LIN {X 0,Y 410.698,Z 448.167,A -85,B 0,C 180,E1 -10512.418,E2 -10512.418} C_VEL
LIN {X 0,Y 412.888,Z 461.606,A -85,B 0,C 180,E1 -10512.911,E2 -10512.911} C_VEL
LIN {X 0,Y 414.693,Z 474.348,A -85,B 0,C 180,E1 -10513.572,E2 -10513.572} C_VEL
LIN {X 0,Y 414.738,Z 479.778,A -85,B 0,C 180,E1 -10513.89,E2 -10513.89} C_VEL
LIN {X 0,Y 413.947,Z 492.112,A -85,B 0,C 180,E1 -10514.742,E2 -10514.742} C_VEL
LIN {X 0,Y 413.113,Z 503.369,A -85,B 0,C 180,E1 -10515.743,E2 -10515.743} C_VEL
LIN {X 0,Y 412.398,Z 514.079,A -85,B 0,C 180,E1 -10516.95,E2 -10516.95} C_VEL
LIN {X 0,Y 411.69,Z 522.971,A -85,B 0,C 180,E1 -10518.179,E2 -10518.179} C_VEL
LIN {X 0,Y 411.063,Z 531.654,A -85,B 0,C 180,E1 -10519.658,E2 -10519.658} C_VEL
LIN {X 0,Y 410.622,Z 538.602,A -85,B 0,C 180,E1 -10521.139,E2 -10521.139} C_VEL
LIN {X 0,Y 410.285,Z 544.173,A -85,B 0,C 180,E1 -10522.619,E2 -10522.619} C_VEL
LIN {X 0,Y 410.107,Z 548.549,A -85,B 0,C 180,E1 -10524.098,E2 -10524.098} C_VEL
LIN {X 0,Y 410.096,Z 550.87,A -85,B 0,C 180,E1 -10525.084,E2 -10525.084} C_VEL
LIN {X 0,Y 409.955,Z 552.745,A -85,B 0,C 180,E1 -10526.068,E2 -10526.068} C_VEL
LIN {X 0,Y 410.007,Z 554.16,A -85,B 0,C 180,E1 -10527.052,E2 -10527.052} C_VEL
LIN {X 0,Y 409.988,Z 555.167,A -85,B 0,C 180,E1 -10528.035,E2 -10528.035} C_VEL
LIN {X 0,Y 409.959,Z 555.78,A -85,B 0,C 180,E1 -10529.018,E2 -10529.018} C_VEL
LIN {X 0,Y 409.967,Z 555.999,A -85,B 0,C 180,E1 -10530,E2 -10530} C_VEL
LIN {X 0,Y 409.959,Z 555.781,A -85,B 0,C 180,E1 -10530.982,E2 -10530.982} C_VEL
LIN {X 0,Y 409.988,Z 555.169,A -85,B 0,C 180,E1 -10531.965,E2 -10531.965} C_VEL
LIN {X 0,Y 410.007,Z 554.163,A -85,B 0,C 180,E1 -10532.948,E2 -10532.948} C_VEL
LIN {X 0,Y 409.955,Z 552.749,A -85,B 0,C 180,E1 -10533.932,E2 -10533.932} C_VEL
LIN {X 0,Y 410.108,Z 549.79,A -85,B 0,C 180,E1 -10535.408,E2 -10535.408} C_VEL
LIN {X 0,Y 410.198,Z 545.778,A -85,B 0,C 180,E1 -10536.888,E2 -10536.888} C_VEL
LIN {X 0,Y 410.551,Z 539.622,A -85,B 0,C 180,E1 -10538.615,E2 -10538.615} C_VEL
LIN {X 0,Y 410.993,Z 532.901,A -85,B 0,C 180,E1 -10540.095,E2 -10540.095} C_VEL
LIN {X 0,Y 411.585,Z 524.569,A -85,B 0,C 180,E1 -10541.574,E2 -10541.574} C_VEL
LIN {X 0,Y 412.248,Z 516.038,A -85,B 0,C 180,E1 -10542.804,E2 -10542.804} C_VEL
LIN {X 0,Y 412.983,Z 505.186,A -85,B 0,C 180,E1 -10544.068,E2 -10544.068} C_VEL
LIN {X 0,Y 413.797,Z 493.656,A -85,B 0,C 180,E1 -10545.137,E2 -10545.137} C_VEL
LIN {X 0,Y 414.677,Z 481.764,A -85,B 0,C 180,E1 -10545.986,E2 -10545.986} C_VEL
LIN {X 0,Y 414.863,Z 475.472,A -85,B 0,C 180,E1 -10546.358,E2 -10546.358} C_VEL
LIN {X 0,Y 412.982,Z 462.163,A -85,B 0,C 180,E1 -10547.062,E2 -10547.062} C_VEL
LIN {X 0,Y 410.941,Z 449.743,A -85,B 0,C 180,E1 -10547.537,E2 -10547.537} C_VEL
LIN {X 0,Y 410.707,Z 447.89,A -85,B 0,C 180,E1 -10547.606,E2 -10547.606} C_VEL
LIN {X 0,Y 411.107,Z 439.39,A -85,B 0,C 180,E1 -10551.039,E2 -10551.039} C_VEL
LIN {X 0,Y 411.526,Z 431.551,A -85,B 0,C 180,E1 -10554.197,E2 -10554.197} C_VEL
LIN {X 0,Y 412.048,Z 423.353,A -85,B 0,C 180,E1 -10557.51,E2 -10557.51} C_VEL
LIN {X 0,Y 412.657,Z 414.499,A -85,B 0,C 180,E1 -10561.185,E2 -10561.185} C_VEL
LIN {X 0,Y 413.314,Z 406.352,A -85,B 0,C 180,E1 -10564.725,E2 -10564.725} C_VEL
LIN {X 0,Y 413.431,Z 402.437,A -85,B 0,C 180,E1 -10566.511,E2 -10566.511} C_VEL
LIN {X 0,Y 412.649,Z 397.214,A -85,B 0,C 180,E1 -10569.062,E2 -10569.062} C_VEL
LIN {X 0,Y 411.729,Z 392.058,A -85,B 0,C 180,E1 -10571.737,E2 -10571.737} C_VEL
LIN {X 0,Y 411.206,Z 389.271,A -85,B 0,C 180,E1 -10573.298,E2 -10573.298} C_VEL
LIN {X 0,Y 411.175,Z 389.269,A -85,B 0,C 180,E1 -10576.866,E2 -10576.866} C_VEL
LIN {X 0,Y 411.221,Z 389.266,A -85,B 0,C 180,E1 -10580.271,E2 -10580.271} C_VEL
LIN {X 0,Y 411.198,Z 389.264,A -85,B 0,C 180,E1 -10583.447,E2 -10583.447} C_VEL
LIN {X 0,Y 411.209,Z 389.265,A -85,B 0,C 180,E1 -10586.873,E2 -10586.873} C_VEL
LIN {X 0,Y 411.235,Z 389.261,A -85,B 0,C 180,E1 -10590.644,E2 -10590.644} C_VEL
LIN {X 0,Y 411.24,Z 389.257,A -85,B 0,C 180,E1 -10593.619,E2 -10593.619} C_VEL
LIN {X 0,Y 411.205,Z 389.265,A -85,B 0,C 180,E1 -10596.853,E2 -10596.853} C_VEL
LIN {X 0,Y 411.218,Z 389.261,A -85,B 0,C 180,E1 -10600.05,E2 -10600.05} C_VEL
LIN {X 0,Y 411.266,Z 389.254,A -85,B 0,C 180,E1 -10603.131,E2 -10603.131} C_VEL
LIN {X 0,Y 411.317,Z 389.25,A -85,B 0,C 180,E1 -10606.891,E2 -10606.891} C_VEL
LIN {X 0,Y 411.311,Z 389.252,A -85,B 0,C 180,E1 -10610.162,E2 -10610.162} C_VEL
LIN {X 0,Y 411.464,Z 389.23,A -85,B 0,C 180,E1 -10613.133,E2 -10613.133} C_VEL
LIN {X 0,Y 411.313,Z 389.248,A -85,B 0,C 180,E1 -10615.099,E2 -10615.099} C_VEL
LIN {X 0,Y 411.515,Z 389.225,A -85,B 0,C 180,E1 -10618.043,E2 -10618.043} C_VEL
LIN {X 0,Y 411.646,Z 389.209,A -85,B 0,C 180,E1 -10620,E2 -10620} C_VEL
LIN {X 0,Y 411.46,Z 389.231,A -85,B 0,C 180,E1 -10622.937,E2 -10622.937} C_VEL
LIN {X 0,Y 411.464,Z 389.23,A -85,B 0,C 180,E1 -10626.867,E2 -10626.867} C_VEL
LIN {X 0,Y 411.295,Z 389.252,A -85,B 0,C 180,E1 -10629.839,E2 -10629.839} C_VEL
LIN {X 0,Y 411.309,Z 389.248,A -85,B 0,C 180,E1 -10633.104,E2 -10633.104} C_VEL
LIN {X 0,Y 411.266,Z 389.254,A -85,B 0,C 180,E1 -10636.869,E2 -10636.869} C_VEL
LIN {X 0,Y 411.234,Z 389.262,A -85,B 0,C 180,E1 -10639.987,E2 -10639.987} C_VEL
LIN {X 0,Y 411.199,Z 389.261,A -85,B 0,C 180,E1 -10643.148,E2 -10643.148} C_VEL
LIN {X 0,Y 411.24,Z 389.259,A -85,B 0,C 180,E1 -10646.381,E2 -10646.381} C_VEL
LIN {X 0,Y 411.203,Z 389.266,A -85,B 0,C 180,E1 -10649.713,E2 -10649.713} C_VEL
LIN {X 0,Y 411.209,Z 389.261,A -85,B 0,C 180,E1 -10653.156,E2 -10653.156} C_VEL
LIN {X 0,Y 411.198,Z 389.262,A -85,B 0,C 180,E1 -10656.553,E2 -10656.553} C_VEL
LIN {X 0,Y 411.221,Z 389.264,A -85,B 0,C 180,E1 -10659.729,E2 -10659.729} C_VEL
LIN {X 0,Y 411.176,Z 389.266,A -85,B 0,C 180,E1 -10663.134,E2 -10663.134} C_VEL
LIN {X 0,Y 411.235,Z 389.262,A -85,B 0,C 180,E1 -10665.872,E2 -10665.872} C_VEL
LIN {X 0,Y 411.208,Z 389.26,A -85,B 0,C 180,E1 -10668.765,E2 -10668.765} C_VEL
LIN {X 0,Y 411.194,Z 389.265,A -85,B 0,C 180,E1 -10672.026,E2 -10672.026} C_VEL
LIN {X 0,Y 411.078,Z 389.28,A -85,B 0,C 180,E1 -10675.149,E2 -10675.149} C_VEL
LIN {X 0,Y 410.745,Z 389.323,A -85,B 0,C 180,E1 -10677.966,E2 -10677.966} C_VEL
LIN {X 0,Y 410.663,Z 389.786,A -85,B 0,C 180,E1 -10679.108,E2 -10679.108} C_VEL
LIN {X 0,Y 410.601,Z 391.828,A -85,B 0,C 180,E1 -10681.363,E2 -10681.363} C_VEL
LIN {X 0,Y 410.51,Z 394.919,A -85,B 0,C 180,E1 -10684.659,E2 -10684.659} C_VEL
LIN {X 0,Y 410.426,Z 398.086,A -85,B 0,C 180,E1 -10687.869,E2 -10687.869} C_VEL
LIN {X 0,Y 410.399,Z 401.392,A -85,B 0,C 180,E1 -10691.012,E2 -10691.012} C_VEL
LIN {X 0,Y 410.37,Z 403.05,A -85,B 0,C 180,E1 -10692.502,E2 -10692.502} C_VEL
LIN {X 0,Y 414.194,Z 417.585,A -85,B 0,C 180,E1 -10693.187,E2 -10693.187} C_VEL
LIN {X 0,Y 415.645,Z 424.633,A -85,B 0,C 180,E1 -10693.592,E2 -10693.592} C_VEL
LIN {X 0,Y 415.134,Z 436.175,A -85,B 0,C 180,E1 -10694.284,E2 -10694.284} C_VEL
LIN {X 0,Y 414.53,Z 446.816,A -85,B 0,C 180,E1 -10695.103,E2 -10695.103} C_VEL
LIN {X 0,Y 413.752,Z 458.523,A -85,B 0,C 180,E1 -10696.243,E2 -10696.243} C_VEL
LIN {X 0,Y 412.944,Z 468.466,A -85,B 0,C 180,E1 -10697.467,E2 -10697.467} C_VEL
LIN {X 0,Y 412.186,Z 478.066,A -85,B 0,C 180,E1 -10698.941,E2 -10698.941} C_VEL
LIN {X 0,Y 411.551,Z 485.722,A -85,B 0,C 180,E1 -10700.416,E2 -10700.416} C_VEL
LIN {X 0,Y 410.968,Z 492.741,A -85,B 0,C 180,E1 -10702.137,E2 -10702.137} C_VEL
LIN {X 0,Y 410.668,Z 497.411,A -85,B 0,C 180,E1 -10703.613,E2 -10703.613} C_VEL
LIN {X 0,Y 410.353,Z 500.99,A -85,B 0,C 180,E1 -10705.088,E2 -10705.088} C_VEL
LIN {X 0,Y 410.376,Z 502.829,A -85,B 0,C 180,E1 -10706.072,E2 -10706.072} C_VEL
LIN {X 0,Y 410.261,Z 504.221,A -85,B 0,C 180,E1 -10707.054,E2 -10707.054} C_VEL
LIN {X 0,Y 410.072,Z 505.825,A -85,B 0,C 180,E1 -10709.018,E2 -10709.018} C_VEL
LIN {X 0,Y 410.065,Z 506.056,A -85,B 0,C 180,E1 -10710,E2 -10710} C_VEL
LIN {X 0,Y 410.148,Z 505.287,A -85,B 0,C 180,E1 -10711.964,E2 -10711.964} C_VEL
LIN {X 0,Y 410.375,Z 502.977,A -85,B 0,C 180,E1 -10713.928,E2 -10713.928} C_VEL
LIN {X 0,Y 410.369,Z 500.144,A -85,B 0,C 180,E1 -10715.405,E2 -10715.405} C_VEL
LIN {X 0,Y 410.733,Z 495.771,A -85,B 0,C 180,E1 -10717.051,E2 -10717.051} C_VEL
LIN {X 0,Y 411.077,Z 491.298,A -85,B 0,C 180,E1 -10718.356,E2 -10718.356} C_VEL
LIN {X 0,Y 411.398,Z 487.566,A -85,B 0,C 180,E1 -10719.267,E2 -10719.267} C_VEL
LIN {X 0,Y 411.046,Z 484.473,A -85,B 0,C 180,E1 -10719.965,E2 -10719.965} C_VEL
LIN {X 0,Y 407.607,Z 476.939,A -85,B 0,C 180,E1 -10721.528,E2 -10721.528} C_VEL
LIN {X 0,Y 406.099,Z 472.057,A -85,B 0,C 180,E1 -10722.379,E2 -10722.379} C_VEL
LIN {X 0,Y 406.011,Z 469.328,A -85,B 0,C 180,E1 -10722.785,E2 -10722.785} C_VEL
LIN {X 0,Y 406.832,Z 459.768,A -85,B 0,C 180,E1 -10723.996,E2 -10723.996} C_VEL
LIN {X 0,Y 407.548,Z 449.017,A -85,B 0,C 180,E1 -10725.095,E2 -10725.095} C_VEL
LIN {X 0,Y 408.242,Z 437.93,A -85,B 0,C 180,E1 -10725.989,E2 -10725.989} C_VEL
LIN {X 0,Y 408.802,Z 426.011,A -85,B 0,C 180,E1 -10726.734,E2 -10726.734} C_VEL
LIN {X 0,Y 406.332,Z 414.61,A -85,B 0,C 180,E1 -10727.395,E2 -10727.395} C_VEL
LIN {X 0,Y 403.3,Z 403.39,A -85,B 0,C 180,E1 -10727.935,E2 -10727.935} C_VEL
LIN {X 0,Y 403.301,Z 400.758,A -85,B 0,C 180,E1 -10730.397,E2 -10730.397} C_VEL
LIN {X 0,Y 403.397,Z 397.5,A -85,B 0,C 180,E1 -10733.623,E2 -10733.623} C_VEL
LIN {X 0,Y 403.481,Z 394.342,A -85,B 0,C 180,E1 -10736.929,E2 -10736.929} C_VEL
LIN {X 0,Y 403.619,Z 391.226,A -85,B 0,C 180,E1 -10740.329,E2 -10740.329} C_VEL
LIN {X 0,Y 403.696,Z 390.202,A -85,B 0,C 180,E1 -10741.485,E2 -10741.485} C_VEL
LIN {X 0,Y 404.044,Z 390.154,A -85,B 0,C 180,E1 -10745.162,E2 -10745.162} C_VEL
LIN {X 0,Y 404.155,Z 390.144,A -85,B 0,C 180,E1 -10748.508,E2 -10748.508} C_VEL
LIN {X 0,Y 404.126,Z 390.142,A -85,B 0,C 180,E1 -10751.6,E2 -10751.6} C_VEL
LIN {X 0,Y 404.148,Z 390.144,A -85,B 0,C 180,E1 -10754.522,E2 -10754.522} C_VEL
LIN {X 0,Y 404.14,Z 390.141,A -85,B 0,C 180,E1 -10757.296,E2 -10757.296} C_VEL
LIN {X 0,Y 404.172,Z 390.14,A -85,B 0,C 180,E1 -10759.956,E2 -10759.956} C_VEL
LIN {X 0,Y 404.144,Z 390.14,A -85,B 0,C 180,E1 -10763.124,E2 -10763.124} C_VEL
LIN {X 0,Y 404.149,Z 390.145,A -85,B 0,C 180,E1 -10766.188,E2 -10766.188} C_VEL
LIN {X 0,Y 404.15,Z 390.142,A -85,B 0,C 180,E1 -10769.715,E2 -10769.715} C_VEL
LIN {X 0,Y 404.199,Z 390.134,A -85,B 0,C 180,E1 -10773.123,E2 -10773.123} C_VEL
LIN {X 0,Y 404.178,Z 390.136,A -85,B 0,C 180,E1 -10775.334,E2 -10775.334} C_VEL
LIN {X 0,Y 404.143,Z 390.142,A -85,B 0,C 180,E1 -10778.581,E2 -10778.581} C_VEL
LIN {X 0,Y 404.213,Z 390.137,A -85,B 0,C 180,E1 -10781.762,E2 -10781.762} C_VEL
LIN {X 0,Y 404.211,Z 390.132,A -85,B 0,C 180,E1 -10784.882,E2 -10784.882} C_VEL
LIN {X 0,Y 404.261,Z 390.132,A -85,B 0,C 180,E1 -10787.959,E2 -10787.959} C_VEL
LIN {X 0,Y 404.27,Z 390.124,A -85,B 0,C 180,E1 -10790.998,E2 -10790.998} C_VEL
LIN {X 0,Y 404.423,Z 390.11,A -85,B 0,C 180,E1 -10794.015,E2 -10794.015} C_VEL
LIN {X 0,Y 404.485,Z 390.102,A -85,B 0,C 180,E1 -10798.008,E2 -10798.008} C_VEL
LIN {X 0,Y 404.614,Z 390.085,A -85,B 0,C 180,E1 -10800,E2 -10800} C_VEL
LIN {X 0,Y 404.42,Z 390.106,A -85,B 0,C 180,E1 -10802.988,E2 -10802.988} C_VEL
LIN {X 0,Y 404.417,Z 390.108,A -85,B 0,C 180,E1 -10806.987,E2 -10806.987} C_VEL
LIN {X 0,Y 404.275,Z 390.126,A -85,B 0,C 180,E1 -10810.011,E2 -10810.011} C_VEL
LIN {X 0,Y 404.271,Z 390.128,A -85,B 0,C 180,E1 -10813.211,E2 -10813.211} C_VEL
LIN {X 0,Y 404.22,Z 390.133,A -85,B 0,C 180,E1 -10817.007,E2 -10817.007} C_VEL
LIN {X 0,Y 404.168,Z 390.138,A -85,B 0,C 180,E1 -10820.351,E2 -10820.351} C_VEL
LIN {X 0,Y 404.172,Z 390.141,A -85,B 0,C 180,E1 -10823.574,E2 -10823.574} C_VEL
LIN {X 0,Y 404.187,Z 390.137,A -85,B 0,C 180,E1 -10825.766,E2 -10825.766} C_VEL
LIN {X 0,Y 404.199,Z 390.133,A -85,B 0,C 180,E1 -10827.999,E2 -10827.999} C_VEL
LIN {X 0,Y 404.143,Z 390.144,A -85,B 0,C 180,E1 -10831.558,E2 -10831.558} C_VEL
LIN {X 0,Y 404.188,Z 390.14,A -85,B 0,C 180,E1 -10835.016,E2 -10835.016} C_VEL
LIN {X 0,Y 404.159,Z 390.142,A -85,B 0,C 180,E1 -10838.757,E2 -10838.757} C_VEL
LIN {X 0,Y 404.126,Z 390.149,A -85,B 0,C 180,E1 -10841.6,E2 -10841.6} C_VEL
LIN {X 0,Y 404.15,Z 390.144,A -85,B 0,C 180,E1 -10844.522,E2 -10844.522} C_VEL
LIN {X 0,Y 404.136,Z 390.161,A -85,B 0,C 180,E1 -10846.378,E2 -10846.378} C_VEL
LIN {X 0,Y 405.308,Z 396.25,A -85,B 0,C 180,E1 -10849.726,E2 -10849.726} C_VEL
LIN {X 0,Y 406.301,Z 402.228,A -85,B 0,C 180,E1 -10852.741,E2 -10852.741} C_VEL
LIN {X 0,Y 406.46,Z 405.637,A -85,B 0,C 180,E1 -10854.357,E2 -10854.357} C_VEL
LIN {X 0,Y 405.815,Z 413.944,A -85,B 0,C 180,E1 -10858.059,E2 -10858.059} C_VEL
LIN {X 0,Y 405.077,Z 423.703,A -85,B 0,C 180,E1 -10862.232,E2 -10862.232} C_VEL
LIN {X 0,Y 404.463,Z 432.528,A -85,B 0,C 180,E1 -10865.899,E2 -10865.899} C_VEL
LIN {X 0,Y 403.964,Z 441.605,A -85,B 0,C 180,E1 -10869.638,E2 -10869.638} C_VEL
LIN {X 0,Y 403.652,Z 447.525,A -85,B 0,C 180,E1 -10872.077,E2 -10872.077} C_VEL
LIN {X 0,Y 406.098,Z 462.801,A -85,B 0,C 180,E1 -10872.684,E2 -10872.684} C_VEL
LIN {X 0,Y 407.872,Z 475.756,A -85,B 0,C 180,E1 -10873.394,E2 -10873.394} C_VEL
LIN {X 0,Y 407.56,Z 485.037,A -85,B 0,C 180,E1 -10873.984,E2 -10873.984} C_VEL
LIN {X 0,Y 406.728,Z 496.091,A -85,B 0,C 180,E1 -10874.85,E2 -10874.85} C_VEL
LIN {X 0,Y 405.874,Z 507.394,A -85,B 0,C 180,E1 -10875.97,E2 -10875.97} C_VEL
LIN {X 0,Y 405.196,Z 517.417,A -85,B 0,C 180,E1 -10877.224,E2 -10877.224} C_VEL
LIN {X 0,Y 404.327,Z 527.131,A -85,B 0,C 180,E1 -10878.723,E2 -10878.723} C_VEL
LIN {X 0,Y 403.782,Z 534.88,A -85,B 0,C 180,E1 -10880.229,E2 -10880.229} C_VEL
LIN {X 0,Y 403.301,Z 542.027,A -85,B 0,C 180,E1 -10881.986,E2 -10881.986} C_VEL
LIN {X 0,Y 403.07,Z 547.241,A -85,B 0,C 180,E1 -10883.65,E2 -10883.65} C_VEL
LIN {X 0,Y 403.009,Z 550.437,A -85,B 0,C 180,E1 -10884.998,E2 -10884.998} C_VEL
LIN {X 0,Y 402.878,Z 552.313,A -85,B 0,C 180,E1 -10885.999,E2 -10885.999} C_VEL
LIN {X 0,Y 402.909,Z 553.727,A -85,B 0,C 180,E1 -10887,E2 -10887} C_VEL
LIN {X 0,Y 402.921,Z 554.736,A -85,B 0,C 180,E1 -10888.001,E2 -10888.001} C_VEL
LIN {X 0,Y 402.884,Z 555.349,A -85,B 0,C 180,E1 -10889,E2 -10889} C_VEL
LIN {X 0,Y 402.89,Z 555.568,A -85,B 0,C 180,E1 -10890,E2 -10890} C_VEL
LIN {X 0,Y 402.884,Z 555.35,A -85,B 0,C 180,E1 -10890.999,E2 -10890.999} C_VEL
LIN {X 0,Y 402.921,Z 554.738,A -85,B 0,C 180,E1 -10891.999,E2 -10891.999} C_VEL
LIN {X 0,Y 402.909,Z 553.731,A -85,B 0,C 180,E1 -10893,E2 -10893} C_VEL
LIN {X 0,Y 402.878,Z 552.317,A -85,B 0,C 180,E1 -10894.001,E2 -10894.001} C_VEL
LIN {X 0,Y 403.006,Z 549.355,A -85,B 0,C 180,E1 -10895.504,E2 -10895.504} C_VEL
LIN {X 0,Y 403.116,Z 545.343,A -85,B 0,C 180,E1 -10897.01,E2 -10897.01} C_VEL
LIN {X 0,Y 403.516,Z 539.188,A -85,B 0,C 180,E1 -10898.766,E2 -10898.766} C_VEL
LIN {X 0,Y 403.965,Z 532.465,A -85,B 0,C 180,E1 -10900.272,E2 -10900.272} C_VEL
LIN {X 0,Y 404.591,Z 524.133,A -85,B 0,C 180,E1 -10901.777,E2 -10901.777} C_VEL
LIN {X 0,Y 405.264,Z 515.6,A -85,B 0,C 180,E1 -10903.029,E2 -10903.029} C_VEL
LIN {X 0,Y 405.98,Z 505.781,A -85,B 0,C 180,E1 -10904.204,E2 -10904.204} C_VEL
LIN {X 0,Y 406.821,Z 494.653,A -85,B 0,C 180,E1 -10905.275,E2 -10905.275} C_VEL
LIN {X 0,Y 407.687,Z 483.364,A -85,B 0,C 180,E1 -10906.131,E2 -10906.131} C_VEL
LIN {X 0,Y 407.882,Z 475.734,A -85,B 0,C 180,E1 -10906.606,E2 -10906.606} C_VEL
LIN {X 0,Y 406.135,Z 462.792,A -85,B 0,C 180,E1 -10907.313,E2 -10907.313} C_VEL
LIN {X 0,Y 403.91,Z 449.366,A -85,B 0,C 180,E1 -10907.85,E2 -10907.85} C_VEL
LIN {X 0,Y 403.658,Z 447.51,A -85,B 0,C 180,E1 -10907.904,E2 -10907.904} C_VEL
LIN {X 0,Y 404.098,Z 439.017,A -85,B 0,C 180,E1 -10911.422,E2 -10911.422} C_VEL
LIN {X 0,Y 404.512,Z 431.208,A -85,B 0,C 180,E1 -10914.644,E2 -10914.644} C_VEL
LIN {X 0,Y 405.094,Z 423.257,A -85,B 0,C 180,E1 -10917.932,E2 -10917.932} C_VEL
LIN {X 0,Y 405.813,Z 413.858,A -85,B 0,C 180,E1 -10921.94,E2 -10921.94} C_VEL
LIN {X 0,Y 406.329,Z 407.41,A -85,B 0,C 180,E1 -10924.805,E2 -10924.805} C_VEL
LIN {X 0,Y 406.447,Z 403.512,A -85,B 0,C 180,E1 -10926.623,E2 -10926.623} C_VEL
LIN {X 0,Y 405.627,Z 398.163,A -85,B 0,C 180,E1 -10929.288,E2 -10929.288} C_VEL
LIN {X 0,Y 404.494,Z 391.852,A -85,B 0,C 180,E1 -10932.658,E2 -10932.658} C_VEL
LIN {X 0,Y 404.127,Z 390.155,A -85,B 0,C 180,E1 -10933.621,E2 -10933.621} C_VEL
LIN {X 0,Y 404.155,Z 390.144,A -85,B 0,C 180,E1 -10936.916,E2 -10936.916} C_VEL
LIN {X 0,Y 404.171,Z 390.141,A -85,B 0,C 180,E1 -10939.955,E2 -10939.955} C_VEL
LIN {X 0,Y 404.142,Z 390.145,A -85,B 0,C 180,E1 -10943.124,E2 -10943.124} C_VEL
LIN {X 0,Y 404.147,Z 390.141,A -85,B 0,C 180,E1 -10946.188,E2 -10946.188} C_VEL
LIN {X 0,Y 404.148,Z 390.139,A -85,B 0,C 180,E1 -10949.715,E2 -10949.715} C_VEL
LIN {X 0,Y 404.197,Z 390.137,A -85,B 0,C 180,E1 -10953.123,E2 -10953.123} C_VEL
LIN {X 0,Y 404.179,Z 390.137,A -85,B 0,C 180,E1 -10955.334,E2 -10955.334} C_VEL
LIN {X 0,Y 404.142,Z 390.145,A -85,B 0,C 180,E1 -10958.581,E2 -10958.581} C_VEL
LIN {X 0,Y 404.214,Z 390.132,A -85,B 0,C 180,E1 -10961.762,E2 -10961.762} C_VEL
LIN {X 0,Y 404.211,Z 390.135,A -85,B 0,C 180,E1 -10964.882,E2 -10964.882} C_VEL
LIN {X 0,Y 404.273,Z 390.126,A -85,B 0,C 180,E1 -10967.959,E2 -10967.959} C_VEL
LIN {X 0,Y 404.437,Z 390.107,A -85,B 0,C 180,E1 -10972.1,E2 -10972.1} C_VEL
LIN {X 0,Y 404.427,Z 390.108,A -85,B 0,C 180,E1 -10974.015,E2 -10974.015} C_VEL
LIN {X 0,Y 404.484,Z 390.1,A -85,B 0,C 180,E1 -10978.009,E2 -10978.009} C_VEL
LIN {X 0,Y 404.615,Z 390.085,A -85,B 0,C 180,E1 -10980,E2 -10980} C_VEL
LIN {X 0,Y 404.418,Z 390.107,A -85,B 0,C 180,E1 -10982.988,E2 -10982.988} C_VEL
LIN {X 0,Y 404.415,Z 390.107,A -85,B 0,C 180,E1 -10986.987,E2 -10986.987} C_VEL
LIN {X 0,Y 404.261,Z 390.13,A -85,B 0,C 180,E1 -10990.012,E2 -10990.012} C_VEL
LIN {X 0,Y 404.269,Z 390.125,A -85,B 0,C 180,E1 -10993.211,E2 -10993.211} C_VEL
LIN {X 0,Y 404.219,Z 390.132,A -85,B 0,C 180,E1 -10997.007,E2 -10997.007} C_VEL
LIN {X 0,Y 404.167,Z 390.141,A -85,B 0,C 180,E1 -11000.352,E2 -11000.352} C_VEL
LIN {X 0,Y 404.166,Z 390.139,A -85,B 0,C 180,E1 -11003.575,E2 -11003.575} C_VEL
LIN {X 0,Y 404.186,Z 390.14,A -85,B 0,C 180,E1 -11005.766,E2 -11005.766} C_VEL
LIN {X 0,Y 404.198,Z 390.138,A -85,B 0,C 180,E1 -11008,E2 -11008} C_VEL
LIN {X 0,Y 404.142,Z 390.144,A -85,B 0,C 180,E1 -11011.558,E2 -11011.558} C_VEL
LIN {X 0,Y 404.188,Z 390.135,A -85,B 0,C 180,E1 -11015.016,E2 -11015.016} C_VEL
LIN {X 0,Y 404.162,Z 390.138,A -85,B 0,C 180,E1 -11018.756,E2 -11018.756} C_VEL
LIN {X 0,Y 404.126,Z 390.148,A -85,B 0,C 180,E1 -11021.6,E2 -11021.6} C_VEL
LIN {X 0,Y 404.156,Z 390.139,A -85,B 0,C 180,E1 -11024.523,E2 -11024.523} C_VEL
LIN {X 0,Y 404.21,Z 390.135,A -85,B 0,C 180,E1 -11027.305,E2 -11027.305} C_VEL
LIN {X 0,Y 404.171,Z 390.14,A -85,B 0,C 180,E1 -11029.955,E2 -11029.955} C_VEL
LIN {X 0,Y 404.12,Z 390.146,A -85,B 0,C 180,E1 -11033.129,E2 -11033.129} C_VEL
LIN {X 0,Y 404.046,Z 390.154,A -85,B 0,C 180,E1 -11034.97,E2 -11034.97} C_VEL
LIN {X 0,Y 403.618,Z 390.211,A -85,B 0,C 180,E1 -11038.563,E2 -11038.563} C_VEL
LIN {X 0,Y 403.598,Z 392.184,A -85,B 0,C 180,E1 -11040.819,E2 -11040.819} C_VEL
LIN {X 0,Y 403.455,Z 395.275,A -85,B 0,C 180,E1 -11044.184,E2 -11044.184} C_VEL
LIN {X 0,Y 403.383,Z 398.468,A -85,B 0,C 180,E1 -11047.462,E2 -11047.462} C_VEL
LIN {X 0,Y 403.365,Z 401.809,A -85,B 0,C 180,E1 -11050.668,E2 -11050.668} C_VEL
LIN {X 0,Y 403.318,Z 403.488,A -85,B 0,C 180,E1 -11052.193,E2 -11052.193} C_VEL
LIN {X 0,Y 406.891,Z 416.983,A -85,B 0,C 180,E1 -11052.83,E2 -11052.83} C_VEL
LIN {X 0,Y 408.773,Z 425.368,A -85,B 0,C 180,E1 -11053.325,E2 -11053.325} C_VEL
LIN {X 0,Y 408.328,Z 436.612,A -85,B 0,C 180,E1 -11054.015,E2 -11054.015} C_VEL
LIN {X 0,Y 407.649,Z 447.828,A -85,B 0,C 180,E1 -11054.898,E2 -11054.898} C_VEL
LIN {X 0,Y 406.894,Z 458.958,A -85,B 0,C 180,E1 -11056.006,E2 -11056.006} C_VEL
LIN {X 0,Y 406.031,Z 468.901,A -85,B 0,C 180,E1 -11057.25,E2 -11057.25} C_VEL
LIN {X 0,Y 405.243,Z 478.5,A -85,B 0,C 180,E1 -11058.749,E2 -11058.749} C_VEL
LIN {X 0,Y 404.567,Z 486.156,A -85,B 0,C 180,E1 -11060.249,E2 -11060.249} C_VEL
LIN {X 0,Y 403.937,Z 493.175,A -85,B 0,C 180,E1 -11061.999,E2 -11061.999} C_VEL
LIN {X 0,Y 403.636,Z 497.843,A -85,B 0,C 180,E1 -11063.502,E2 -11063.502} C_VEL
LIN {X 0,Y 403.279,Z 501.424,A -85,B 0,C 180,E1 -11065.001,E2 -11065.001} C_VEL
LIN {X 0,Y 403.321,Z 503.26,A -85,B 0,C 180,E1 -11066.003,E2 -11066.003} C_VEL
LIN {X 0,Y 403.199,Z 504.653,A -85,B 0,C 180,E1 -11067.003,E2 -11067.003} C_VEL
LIN {X 0,Y 402.993,Z 506.256,A -85,B 0,C 180,E1 -11069.001,E2 -11069.001} C_VEL
LIN {X 0,Y 402.983,Z 506.488,A -85,B 0,C 180,E1 -11070,E2 -11070} C_VEL
LIN {X 0,Y 403.075,Z 505.718,A -85,B 0,C 180,E1 -11071.999,E2 -11071.999} C_VEL
LIN {X 0,Y 403.32,Z 503.407,A -85,B 0,C 180,E1 -11073.997,E2 -11073.997} C_VEL
LIN {X 0,Y 403.32,Z 500.574,A -85,B 0,C 180,E1 -11075.5,E2 -11075.5} C_VEL
LIN {X 0,Y 403.695,Z 496.422,A -85,B 0,C 180,E1 -11077.102,E2 -11077.102} C_VEL
LIN {X 0,Y 404.058,Z 491.728,A -85,B 0,C 180,E1 -11078.502,E2 -11078.502} C_VEL
LIN {X 0,Y 404.665,Z 485.447,A -85,B 0,C 180,E1 -11080.002,E2 -11080.002} C_VEL
LIN {X 0,Y 405.311,Z 477.586,A -85,B 0,C 180,E1 -11081.502,E2 -11081.502} C_VEL
LIN {X 0,Y 406.011,Z 469.328,A -85,B 0,C 180,E1 -11082.785,E2 -11082.785} C_VEL
LIN {X 0,Y 405.692,Z 465.151,A -85,B 0,C 180,E1 -11083.376,E2 -11083.376} C_VEL
LIN {X 0,Y 403.424,Z 458.187,A -85,B 0,C 180,E1 -11084.329,E2 -11084.329} C_VEL
LIN {X 0,Y 401.199,Z 450.764,A -85,B 0,C 180,E1 -11085.209,E2 -11085.209} C_VEL
LIN {X 0,Y 400.935,Z 445.857,A -85,B 0,C 180,E1 -11085.678,E2 -11085.678} C_VEL
LIN {X 0,Y 401.658,Z 435.406,A -85,B 0,C 180,E1 -11086.476,E2 -11086.476} C_VEL
LIN {X 0,Y 402.018,Z 427.154,A -85,B 0,C 180,E1 -11086.983,E2 -11086.983} C_VEL
LIN {X 0,Y 399.399,Z 415.296,A -85,B 0,C 180,E1 -11087.695,E2 -11087.695} C_VEL
LIN {X 0,Y 396.237,Z 403.83,A -85,B 0,C 180,E1 -11088.25,E2 -11088.25} C_VEL
LIN {X 0,Y 396.235,Z 401.161,A -85,B 0,C 180,E1 -11090.778,E2 -11090.778} C_VEL
LIN {X 0,Y 396.373,Z 397.878,A -85,B 0,C 180,E1 -11094.067,E2 -11094.067} C_VEL
LIN {X 0,Y 396.454,Z 394.696,A -85,B 0,C 180,E1 -11097.446,E2 -11097.446} C_VEL
LIN {X 0,Y 396.604,Z 391.531,A -85,B 0,C 180,E1 -11100.924,E2 -11100.924} C_VEL
LIN {X 0,Y 396.686,Z 391.074,A -85,B 0,C 180,E1 -11102.107,E2 -11102.107} C_VEL
LIN {X 0,Y 397.007,Z 391.029,A -85,B 0,C 180,E1 -11105.48,E2 -11105.48} C_VEL
LIN {X 0,Y 397.132,Z 391.016,A -85,B 0,C 180,E1 -11108.861,E2 -11108.861} C_VEL
LIN {X 0,Y 397.072,Z 391.026,A -85,B 0,C 180,E1 -11112.267,E2 -11112.267} C_VEL
LIN {X 0,Y 397.09,Z 391.02,A -85,B 0,C 180,E1 -11115.069,E2 -11115.069} C_VEL
LIN {X 0,Y 397.07,Z 391.025,A -85,B 0,C 180,E1 -11118.021,E2 -11118.021} C_VEL
LIN {X 0,Y 397.138,Z 391.013,A -85,B 0,C 180,E1 -11121.138,E2 -11121.138} C_VEL
LIN {X 0,Y 397.124,Z 391.018,A -85,B 0,C 180,E1 -11124.497,E2 -11124.497} C_VEL
LIN {X 0,Y 397.083,Z 391.024,A -85,B 0,C 180,E1 -11127.929,E2 -11127.929} C_VEL
LIN {X 0,Y 397.126,Z 391.015,A -85,B 0,C 180,E1 -11131.456,E2 -11131.456} C_VEL
LIN {X 0,Y 397.156,Z 391.013,A -85,B 0,C 180,E1 -11134.488,E2 -11134.488} C_VEL
LIN {X 0,Y 397.1,Z 391.022,A -85,B 0,C 180,E1 -11138.182,E2 -11138.182} C_VEL
LIN {X 0,Y 397.165,Z 391.011,A -85,B 0,C 180,E1 -11141.427,E2 -11141.427} C_VEL
LIN {X 0,Y 397.184,Z 391.008,A -85,B 0,C 180,E1 -11144.608,E2 -11144.608} C_VEL
LIN {X 0,Y 397.224,Z 391.007,A -85,B 0,C 180,E1 -11147.742,E2 -11147.742} C_VEL
LIN {X 0,Y 397.24,Z 391,A -85,B 0,C 180,E1 -11150.838,E2 -11150.838} C_VEL
LIN {X 0,Y 397.373,Z 390.988,A -85,B 0,C 180,E1 -11153.908,E2 -11153.908} C_VEL
LIN {X 0,Y 397.454,Z 390.978,A -85,B 0,C 180,E1 -11157.973,E2 -11157.973} C_VEL
LIN {X 0,Y 397.584,Z 390.961,A -85,B 0,C 180,E1 -11160,E2 -11160} C_VEL
LIN {X 0,Y 397.379,Z 390.983,A -85,B 0,C 180,E1 -11163.041,E2 -11163.041} C_VEL
LIN {X 0,Y 397.369,Z 390.986,A -85,B 0,C 180,E1 -11167.112,E2 -11167.112} C_VEL
LIN {X 0,Y 397.233,Z 391.002,A -85,B 0,C 180,E1 -11170.191,E2 -11170.191} C_VEL
LIN {X 0,Y 397.231,Z 391.006,A -85,B 0,C 180,E1 -11173.321,E2 -11173.321} C_VEL
LIN {X 0,Y 397.186,Z 391.01,A -85,B 0,C 180,E1 -11177.155,E2 -11177.155} C_VEL
LIN {X 0,Y 397.107,Z 391.018,A -85,B 0,C 180,E1 -11180.73,E2 -11180.73} C_VEL
LIN {X 0,Y 397.136,Z 391.014,A -85,B 0,C 180,E1 -11184.018,E2 -11184.018} C_VEL
LIN {X 0,Y 397.198,Z 391.01,A -85,B 0,C 180,E1 -11187.39,E2 -11187.39} C_VEL
LIN {X 0,Y 397.083,Z 391.023,A -85,B 0,C 180,E1 -11190.882,E2 -11190.882} C_VEL
LIN {X 0,Y 397.129,Z 391.015,A -85,B 0,C 180,E1 -11194.493,E2 -11194.493} C_VEL
LIN {X 0,Y 397.107,Z 391.017,A -85,B 0,C 180,E1 -11198.275,E2 -11198.275} C_VEL
LIN {X 0,Y 397.092,Z 391.023,A -85,B 0,C 180,E1 -11200.908,E2 -11200.908} C_VEL
LIN {X 0,Y 397.104,Z 391.023,A -85,B 0,C 180,E1 -11203.648,E2 -11203.648} C_VEL
LIN {X 0,Y 397.115,Z 391.062,A -85,B 0,C 180,E1 -11206.002,E2 -11206.002} C_VEL
LIN {X 0,Y 398.243,Z 397.069,A -85,B 0,C 180,E1 -11209.363,E2 -11209.363} C_VEL
LIN {X 0,Y 399.229,Z 402.864,A -85,B 0,C 180,E1 -11212.39,E2 -11212.39} C_VEL
LIN {X 0,Y 399.446,Z 407.233,A -85,B 0,C 180,E1 -11214.506,E2 -11214.506} C_VEL
LIN {X 0,Y 398.781,Z 415.117,A -85,B 0,C 180,E1 -11218.081,E2 -11218.081} C_VEL
LIN {X 0,Y 398.08,Z 424.019,A -85,B 0,C 180,E1 -11221.975,E2 -11221.975} C_VEL
LIN {X 0,Y 397.459,Z 432.183,A -85,B 0,C 180,E1 -11225.447,E2 -11225.447} C_VEL
LIN {X 0,Y 396.938,Z 441.221,A -85,B 0,C 180,E1 -11229.261,E2 -11229.261} C_VEL
LIN {X 0,Y 396.611,Z 447.16,A -85,B 0,C 180,E1 -11231.768,E2 -11231.768} C_VEL
LIN {X 0,Y 398.838,Z 460.535,A -85,B 0,C 180,E1 -11232.282,E2 -11232.282} C_VEL
LIN {X 0,Y 400.678,Z 473.868,A -85,B 0,C 180,E1 -11233.004,E2 -11233.004} C_VEL
LIN {X 0,Y 401.039,Z 479.594,A -85,B 0,C 180,E1 -11233.368,E2 -11233.368} C_VEL
LIN {X 0,Y 400.178,Z 491.248,A -85,B 0,C 180,E1 -11234.204,E2 -11234.204} C_VEL
LIN {X 0,Y 399.27,Z 502.746,A -85,B 0,C 180,E1 -11235.265,E2 -11235.265} C_VEL
LIN {X 0,Y 398.486,Z 513.323,A -85,B 0,C 180,E1 -11236.5,E2 -11236.5} C_VEL
LIN {X 0,Y 397.752,Z 522.107,A -85,B 0,C 180,E1 -11237.758,E2 -11237.758} C_VEL
LIN {X 0,Y 396.982,Z 530.784,A -85,B 0,C 180,E1 -11239.287,E2 -11239.287} C_VEL
LIN {X 0,Y 396.498,Z 537.732,A -85,B 0,C 180,E1 -11240.82,E2 -11240.82} C_VEL
LIN {X 0,Y 396.14,Z 543.305,A -85,B 0,C 180,E1 -11242.353,E2 -11242.353} C_VEL
LIN {X 0,Y 395.95,Z 547.683,A -85,B 0,C 180,E1 -11243.886,E2 -11243.886} C_VEL
LIN {X 0,Y 395.922,Z 550.005,A -85,B 0,C 180,E1 -11244.908,E2 -11244.908} C_VEL
LIN {X 0,Y 395.803,Z 551.881,A -85,B 0,C 180,E1 -11245.927,E2 -11245.927} C_VEL
LIN {X 0,Y 395.813,Z 553.295,A -85,B 0,C 180,E1 -11246.946,E2 -11246.946} C_VEL
LIN {X 0,Y 395.854,Z 554.305,A -85,B 0,C 180,E1 -11247.965,E2 -11247.965} C_VEL
LIN {X 0,Y 395.813,Z 554.918,A -85,B 0,C 180,E1 -11248.982,E2 -11248.982} C_VEL
LIN {X 0,Y 395.815,Z 555.137,A -85,B 0,C 180,E1 -11250,E2 -11250} C_VEL
LIN {X 0,Y 395.813,Z 554.919,A -85,B 0,C 180,E1 -11251.017,E2 -11251.017} C_VEL
LIN {X 0,Y 395.854,Z 554.307,A -85,B 0,C 180,E1 -11252.035,E2 -11252.035} C_VEL
LIN {X 0,Y 395.813,Z 553.297,A -85,B 0,C 180,E1 -11253.053,E2 -11253.053} C_VEL
LIN {X 0,Y 395.802,Z 551.884,A -85,B 0,C 180,E1 -11254.073,E2 -11254.073} C_VEL
LIN {X 0,Y 395.907,Z 548.92,A -85,B 0,C 180,E1 -11255.603,E2 -11255.603} C_VEL
LIN {X 0,Y 396.061,Z 544.909,A -85,B 0,C 180,E1 -11257.135,E2 -11257.135} C_VEL
LIN {X 0,Y 396.458,Z 538.752,A -85,B 0,C 180,E1 -11258.923,E2 -11258.923} C_VEL
LIN {X 0,Y 396.914,Z 532.027,A -85,B 0,C 180,E1 -11260.457,E2 -11260.457} C_VEL
LIN {X 0,Y 397.582,Z 523.695,A -85,B 0,C 180,E1 -11261.988,E2 -11261.988} C_VEL
LIN {X 0,Y 398.304,Z 515.163,A -85,B 0,C 180,E1 -11263.261,E2 -11263.261} C_VEL
LIN {X 0,Y 399.102,Z 504.865,A -85,B 0,C 180,E1 -11264.507,E2 -11264.507} C_VEL
LIN {X 0,Y 399.954,Z 494.216,A -85,B 0,C 180,E1 -11265.544,E2 -11265.544} C_VEL
LIN {X 0,Y 400.859,Z 483.018,A -85,B 0,C 180,E1 -11266.407,E2 -11266.407} C_VEL
LIN {X 0,Y 401.112,Z 477.794,A -85,B 0,C 180,E1 -11266.745,E2 -11266.745} C_VEL
LIN {X 0,Y 399.448,Z 465.095,A -85,B 0,C 180,E1 -11267.495,E2 -11267.495} C_VEL
LIN {X 0,Y 397.417,Z 452.01,A -85,B 0,C 180,E1 -11268.066,E2 -11268.066} C_VEL
LIN {X 0,Y 396.61,Z 447.109,A -85,B 0,C 180,E1 -11268.232,E2 -11268.232} C_VEL
LIN {X 0,Y 397.073,Z 438.645,A -85,B 0,C 180,E1 -11271.82,E2 -11271.82} C_VEL
LIN {X 0,Y 397.518,Z 430.86,A -85,B 0,C 180,E1 -11275.107,E2 -11275.107} C_VEL
LIN {X 0,Y 398.128,Z 422.958,A -85,B 0,C 180,E1 -11278.465,E2 -11278.465} C_VEL
LIN {X 0,Y 398.827,Z 414.303,A -85,B 0,C 180,E1 -11282.238,E2 -11282.238} C_VEL
LIN {X 0,Y 399.444,Z 407.164,A -85,B 0,C 180,E1 -11285.494,E2 -11285.494} C_VEL
LIN {X 0,Y 399.222,Z 402.845,A -85,B 0,C 180,E1 -11287.609,E2 -11287.609} C_VEL
LIN {X 0,Y 398.169,Z 396.796,A -85,B 0,C 180,E1 -11290.774,E2 -11290.774} C_VEL
LIN {X 0,Y 397.124,Z 391.026,A -85,B 0,C 180,E1 -11294.085,E2 -11294.085} C_VEL
LIN {X 0,Y 397.104,Z 391.021,A -85,B 0,C 180,E1 -11296.521,E2 -11296.521} C_VEL
LIN {X 0,Y 397.117,Z 391.022,A -85,B 0,C 180,E1 -11300.423,E2 -11300.423} C_VEL
LIN {X 0,Y 397.112,Z 391.018,A -85,B 0,C 180,E1 -11304.266,E2 -11304.266} C_VEL
LIN {X 0,Y 397.117,Z 391.02,A -85,B 0,C 180,E1 -11306.727,E2 -11306.727} C_VEL
LIN {X 0,Y 397.127,Z 391.016,A -85,B 0,C 180,E1 -11310.296,E2 -11310.296} C_VEL
LIN {X 0,Y 397.197,Z 391.01,A -85,B 0,C 180,E1 -11312.61,E2 -11312.61} C_VEL
LIN {X 0,Y 397.135,Z 391.014,A -85,B 0,C 180,E1 -11315.982,E2 -11315.982} C_VEL
LIN {X 0,Y 397.141,Z 391.013,A -85,B 0,C 180,E1 -11319.705,E2 -11319.705} C_VEL
LIN {X 0,Y 397.185,Z 391.011,A -85,B 0,C 180,E1 -11322.845,E2 -11322.845} C_VEL
LIN {X 0,Y 397.229,Z 391.006,A -85,B 0,C 180,E1 -11326.679,E2 -11326.679} C_VEL
LIN {X 0,Y 397.232,Z 391.002,A -85,B 0,C 180,E1 -11329.809,E2 -11329.809} C_VEL
LIN {X 0,Y 397.368,Z 390.987,A -85,B 0,C 180,E1 -11332.888,E2 -11332.888} C_VEL
LIN {X 0,Y 397.257,Z 391,A -85,B 0,C 180,E1 -11334.925,E2 -11334.925} C_VEL
LIN {X 0,Y 397.453,Z 390.976,A -85,B 0,C 180,E1 -11337.973,E2 -11337.973} C_VEL
LIN {X 0,Y 397.585,Z 390.96,A -85,B 0,C 180,E1 -11340,E2 -11340} C_VEL
LIN {X 0,Y 397.378,Z 390.984,A -85,B 0,C 180,E1 -11343.041,E2 -11343.041} C_VEL
LIN {X 0,Y 397.368,Z 390.984,A -85,B 0,C 180,E1 -11347.112,E2 -11347.112} C_VEL
LIN {X 0,Y 397.22,Z 391.009,A -85,B 0,C 180,E1 -11350.191,E2 -11350.191} C_VEL
LIN {X 0,Y 397.23,Z 391.002,A -85,B 0,C 180,E1 -11353.321,E2 -11353.321} C_VEL
LIN {X 0,Y 397.185,Z 391.007,A -85,B 0,C 180,E1 -11357.155,E2 -11357.155} C_VEL
LIN {X 0,Y 397.106,Z 391.017,A -85,B 0,C 180,E1 -11360.73,E2 -11360.73} C_VEL
LIN {X 0,Y 397.131,Z 391.019,A -85,B 0,C 180,E1 -11364.019,E2 -11364.019} C_VEL
LIN {X 0,Y 397.197,Z 391.007,A -85,B 0,C 180,E1 -11367.39,E2 -11367.39} C_VEL
LIN {X 0,Y 397.081,Z 391.02,A -85,B 0,C 180,E1 -11370.882,E2 -11370.882} C_VEL
LIN {X 0,Y 397.128,Z 391.015,A -85,B 0,C 180,E1 -11374.493,E2 -11374.493} C_VEL
LIN {X 0,Y 397.11,Z 391.018,A -85,B 0,C 180,E1 -11378.274,E2 -11378.274} C_VEL
LIN {X 0,Y 397.092,Z 391.019,A -85,B 0,C 180,E1 -11380.909,E2 -11380.909} C_VEL
LIN {X 0,Y 397.105,Z 391.022,A -85,B 0,C 180,E1 -11383.648,E2 -11383.648} C_VEL
LIN {X 0,Y 397.164,Z 391.01,A -85,B 0,C 180,E1 -11386.512,E2 -11386.512} C_VEL
LIN {X 0,Y 397.118,Z 391.021,A -85,B 0,C 180,E1 -11389.552,E2 -11389.552} C_VEL
LIN {X 0,Y 397.083,Z 391.02,A -85,B 0,C 180,E1 -11392.794,E2 -11392.794} C_VEL
LIN {X 0,Y 396.918,Z 391.046,A -85,B 0,C 180,E1 -11395.486,E2 -11395.486} C_VEL
LIN {X 0,Y 396.597,Z 391.085,A -85,B 0,C 180,E1 -11398.277,E2 -11398.277} C_VEL
LIN {X 0,Y 396.537,Z 392.482,A -85,B 0,C 180,E1 -11400.247,E2 -11400.247} C_VEL
LIN {X 0,Y 396.425,Z 395.632,A -85,B 0,C 180,E1 -11403.691,E2 -11403.691} C_VEL
LIN {X 0,Y 396.322,Z 399.054,A -85,B 0,C 180,E1 -11407.239,E2 -11407.239} C_VEL
LIN {X 0,Y 396.289,Z 402.208,A -85,B 0,C 180,E1 -11410.308,E2 -11410.308} C_VEL
LIN {X 0,Y 396.266,Z 403.891,A -85,B 0,C 180,E1 -11411.862,E2 -11411.862} C_VEL
LIN {X 0,Y 399.868,Z 417.218,A -85,B 0,C 180,E1 -11412.509,E2 -11412.509} C_VEL
LIN {X 0,Y 401.881,Z 426.13,A -85,B 0,C 180,E1 -11413.048,E2 -11413.048} C_VEL
LIN {X 0,Y 401.652,Z 435.694,A -85,B 0,C 180,E1 -11413.642,E2 -11413.642} C_VEL
LIN {X 0,Y 400.92,Z 446.989,A -85,B 0,C 180,E1 -11414.521,E2 -11414.521} C_VEL
LIN {X 0,Y 400.22,Z 457.546,A -85,B 0,C 180,E1 -11415.562,E2 -11415.562} C_VEL
LIN {X 0,Y 399.296,Z 467.532,A -85,B 0,C 180,E1 -11416.773,E2 -11416.773} C_VEL
LIN {X 0,Y 398.573,Z 475.991,A -85,B 0,C 180,E1 -11418.042,E2 -11418.042} C_VEL
LIN {X 0,Y 397.836,Z 484.203,A -85,B 0,C 180,E1 -11419.568,E2 -11419.568} C_VEL
LIN {X 0,Y 397.257,Z 489.823,A -85,B 0,C 180,E1 -11420.838,E2 -11420.838} C_VEL
LIN {X 0,Y 396.807,Z 495.293,A -85,B 0,C 180,E1 -11422.367,E2 -11422.367} C_VEL
LIN {X 0,Y 396.435,Z 499.585,A -85,B 0,C 180,E1 -11423.894,E2 -11423.894} C_VEL
LIN {X 0,Y 396.211,Z 501.857,A -85,B 0,C 180,E1 -11424.912,E2 -11424.912} C_VEL
LIN {X 0,Y 396.247,Z 503.693,A -85,B 0,C 180,E1 -11425.932,E2 -11425.932} C_VEL
LIN {X 0,Y 396.14,Z 505.084,A -85,B 0,C 180,E1 -11426.949,E2 -11426.949} C_VEL
LIN {X 0,Y 395.917,Z 506.687,A -85,B 0,C 180,E1 -11428.983,E2 -11428.983} C_VEL
LIN {X 0,Y 395.904,Z 506.919,A -85,B 0,C 180,E1 -11430,E2 -11430} C_VEL
LIN {X 0,Y 396.005,Z 506.148,A -85,B 0,C 180,E1 -11432.034,E2 -11432.034} C_VEL
LIN {X 0,Y 396.133,Z 505.185,A -85,B 0,C 180,E1 -11433.051,E2 -11433.051} C_VEL
LIN {X 0,Y 396.246,Z 503.838,A -85,B 0,C 180,E1 -11434.068,E2 -11434.068} C_VEL
LIN {X 0,Y 396.276,Z 501.004,A -85,B 0,C 180,E1 -11435.598,E2 -11435.598} C_VEL
LIN {X 0,Y 396.633,Z 497.141,A -85,B 0,C 180,E1 -11437.125,E2 -11437.125} C_VEL
LIN {X 0,Y 397.059,Z 492.158,A -85,B 0,C 180,E1 -11438.653,E2 -11438.653} C_VEL
LIN {X 0,Y 397.695,Z 485.876,A -85,B 0,C 180,E1 -11440.179,E2 -11440.179} C_VEL
LIN {X 0,Y 398.36,Z 478.015,A -85,B 0,C 180,E1 -11441.706,E2 -11441.706} C_VEL
LIN {X 0,Y 399.25,Z 468.226,A -85,B 0,C 180,E1 -11443.229,E2 -11443.229} C_VEL
LIN {X 0,Y 400.125,Z 458.566,A -85,B 0,C 180,E1 -11444.425,E2 -11444.425} C_VEL
LIN {X 0,Y 400.816,Z 447.756,A -85,B 0,C 180,E1 -11445.51,E2 -11445.51} C_VEL
LIN {X 0,Y 400.935,Z 445.857,A -85,B 0,C 180,E1 -11445.678,E2 -11445.678} C_VEL
LIN {X 0,Y 400.667,Z 440.793,A -85,B 0,C 180,E1 -11446.119,E2 -11446.119} C_VEL
LIN {X 0,Y 399.389,Z 435.829,A -85,B 0,C 180,E1 -11446.557,E2 -11446.557} C_VEL
LIN {X 0,Y 394.225,Z 422.453,A -85,B 0,C 180,E1 -11447.62,E2 -11447.62} C_VEL
LIN {X 0,Y 393.19,Z 418.866,A -85,B 0,C 180,E1 -11447.843,E2 -11447.843} C_VEL
LIN {X 0,Y 389.613,Z 406.129,A -85,B 0,C 180,E1 -11448.502,E2 -11448.502} C_VEL
LIN {X 0,Y 389.176,Z 404.254,A -85,B 0,C 180,E1 -11448.593,E2 -11448.593} C_VEL
LIN {X 0,Y 389.196,Z 401.564,A -85,B 0,C 180,E1 -11451.171,E2 -11451.171} C_VEL
LIN {X 0,Y 389.318,Z 398.255,A -85,B 0,C 180,E1 -11454.532,E2 -11454.532} C_VEL
LIN {X 0,Y 389.401,Z 395.051,A -85,B 0,C 180,E1 -11457.986,E2 -11457.986} C_VEL
LIN {X 0,Y 389.529,Z 392.917,A -85,B 0,C 180,E1 -11460.344,E2 -11460.344} C_VEL
LIN {X 0,Y 389.591,Z 391.959,A -85,B 0,C 180,E1 -11461.544,E2 -11461.544} C_VEL
LIN {X 0,Y 389.926,Z 391.912,A -85,B 0,C 180,E1 -11465.224,E2 -11465.224} C_VEL
LIN {X 0,Y 390.041,Z 391.897,A -85,B 0,C 180,E1 -11467.781,E2 -11467.781} C_VEL
LIN {X 0,Y 390.059,Z 391.897,A -85,B 0,C 180,E1 -11470.821,E2 -11470.821} C_VEL
LIN {X 0,Y 390.058,Z 391.896,A -85,B 0,C 180,E1 -11473.886,E2 -11473.886} C_VEL
LIN {X 0,Y 390.06,Z 391.897,A -85,B 0,C 180,E1 -11476.79,E2 -11476.79} C_VEL
LIN {X 0,Y 390.061,Z 391.895,A -85,B 0,C 180,E1 -11479.561,E2 -11479.561} C_VEL
LIN {X 0,Y 390.05,Z 391.9,A -85,B 0,C 180,E1 -11482.449,E2 -11482.449} C_VEL
LIN {X 0,Y 390.088,Z 391.896,A -85,B 0,C 180,E1 -11486.047,E2 -11486.047} C_VEL
LIN {X 0,Y 390.051,Z 391.899,A -85,B 0,C 180,E1 -11489.869,E2 -11489.869} C_VEL
LIN {X 0,Y 390.117,Z 391.887,A -85,B 0,C 180,E1 -11493.232,E2 -11493.232} C_VEL
LIN {X 0,Y 390.072,Z 391.893,A -85,B 0,C 180,E1 -11496.764,E2 -11496.764} C_VEL
LIN {X 0,Y 390.108,Z 391.894,A -85,B 0,C 180,E1 -11499.983,E2 -11499.983} C_VEL
LIN {X 0,Y 390.142,Z 391.885,A -85,B 0,C 180,E1 -11503.248,E2 -11503.248} C_VEL
LIN {X 0,Y 390.199,Z 391.878,A -85,B 0,C 180,E1 -11506.562,E2 -11506.562} C_VEL
LIN {X 0,Y 390.172,Z 391.884,A -85,B 0,C 180,E1 -11509.623,E2 -11509.623} C_VEL
LIN {X 0,Y 390.289,Z 391.866,A -85,B 0,C 180,E1 -11512.759,E2 -11512.759} C_VEL
LIN {X 0,Y 390.229,Z 391.874,A -85,B 0,C 180,E1 -11514.833,E2 -11514.833} C_VEL
LIN {X 0,Y 390.422,Z 391.854,A -85,B 0,C 180,E1 -11517.937,E2 -11517.937} C_VEL
LIN {X 0,Y 390.553,Z 391.836,A -85,B 0,C 180,E1 -11520,E2 -11520} C_VEL
LIN {X 0,Y 390.314,Z 391.864,A -85,B 0,C 180,E1 -11523.096,E2 -11523.096} C_VEL
LIN {X 0,Y 390.335,Z 391.861,A -85,B 0,C 180,E1 -11526.202,E2 -11526.202} C_VEL
LIN {X 0,Y 390.32,Z 391.863,A -85,B 0,C 180,E1 -11528.282,E2 -11528.282} C_VEL
LIN {X 0,Y 390.183,Z 391.879,A -85,B 0,C 180,E1 -11532.483,E2 -11532.483} C_VEL
LIN {X 0,Y 390.144,Z 391.888,A -85,B 0,C 180,E1 -11535.677,E2 -11535.677} C_VEL
LIN {X 0,Y 390.109,Z 391.89,A -85,B 0,C 180,E1 -11538.922,E2 -11538.922} C_VEL
LIN {X 0,Y 390.044,Z 391.897,A -85,B 0,C 180,E1 -11542.234,E2 -11542.234} C_VEL
LIN {X 0,Y 390.123,Z 391.889,A -85,B 0,C 180,E1 -11545.743,E2 -11545.743} C_VEL
LIN {X 0,Y 390.063,Z 391.899,A -85,B 0,C 180,E1 -11549.109,E2 -11549.109} C_VEL
LIN {X 0,Y 390.046,Z 391.898,A -85,B 0,C 180,E1 -11552.721,E2 -11552.721} C_VEL
LIN {X 0,Y 390.06,Z 391.895,A -85,B 0,C 180,E1 -11555.825,E2 -11555.825} C_VEL
LIN {X 0,Y 390.074,Z 391.898,A -85,B 0,C 180,E1 -11559.218,E2 -11559.218} C_VEL
LIN {X 0,Y 390.046,Z 391.904,A -85,B 0,C 180,E1 -11562.374,E2 -11562.374} C_VEL
LIN {X 0,Y 390.103,Z 392.075,A -85,B 0,C 180,E1 -11565.684,E2 -11565.684} C_VEL
LIN {X 0,Y 391.155,Z 397.82,A -85,B 0,C 180,E1 -11568.993,E2 -11568.993} C_VEL
LIN {X 0,Y 392.179,Z 403.532,A -85,B 0,C 180,E1 -11572.045,E2 -11572.045} C_VEL
LIN {X 0,Y 392.489,Z 406.984,A -85,B 0,C 180,E1 -11573.778,E2 -11573.778} C_VEL
LIN {X 0,Y 392.088,Z 412.214,A -85,B 0,C 180,E1 -11576.243,E2 -11576.243} C_VEL
LIN {X 0,Y 391.622,Z 417.449,A -85,B 0,C 180,E1 -11578.638,E2 -11578.638} C_VEL
LIN {X 0,Y 390.976,Z 425.31,A -85,B 0,C 180,E1 -11582.136,E2 -11582.136} C_VEL
LIN {X 0,Y 390.374,Z 433.13,A -85,B 0,C 180,E1 -11585.539,E2 -11585.539} C_VEL
LIN {X 0,Y 389.907,Z 440.832,A -85,B 0,C 180,E1 -11588.869,E2 -11588.869} C_VEL
LIN {X 0,Y 389.569,Z 446.744,A -85,B 0,C 180,E1 -11591.426,E2 -11591.426} C_VEL
LIN {X 0,Y 391.86,Z 460.659,A -85,B 0,C 180,E1 -11591.979,E2 -11591.979} C_VEL
LIN {X 0,Y 393.656,Z 474.09,A -85,B 0,C 180,E1 -11592.73,E2 -11592.73} C_VEL
LIN {X 0,Y 394.175,Z 479.454,A -85,B 0,C 180,E1 -11593.089,E2 -11593.089} C_VEL
LIN {X 0,Y 393.346,Z 490.819,A -85,B 0,C 180,E1 -11593.922,E2 -11593.922} C_VEL
LIN {X 0,Y 392.408,Z 501.84,A -85,B 0,C 180,E1 -11594.948,E2 -11594.948} C_VEL
LIN {X 0,Y 391.683,Z 511.49,A -85,B 0,C 180,E1 -11596.072,E2 -11596.072} C_VEL
LIN {X 0,Y 390.801,Z 521.675,A -85,B 0,C 180,E1 -11597.537,E2 -11597.537} C_VEL
LIN {X 0,Y 389.965,Z 530.35,A -85,B 0,C 180,E1 -11599.092,E2 -11599.092} C_VEL
LIN {X 0,Y 389.453,Z 537.299,A -85,B 0,C 180,E1 -11600.653,E2 -11600.653} C_VEL
LIN {X 0,Y 389.078,Z 542.872,A -85,B 0,C 180,E1 -11602.214,E2 -11602.214} C_VEL
LIN {X 0,Y 388.834,Z 548.024,A -85,B 0,C 180,E1 -11604.094,E2 -11604.094} C_VEL
LIN {X 0,Y 388.73,Z 551.45,A -85,B 0,C 180,E1 -11605.853,E2 -11605.853} C_VEL
LIN {X 0,Y 388.788,Z 553.875,A -85,B 0,C 180,E1 -11607.928,E2 -11607.928} C_VEL
LIN {X 0,Y 388.743,Z 554.488,A -85,B 0,C 180,E1 -11608.964,E2 -11608.964} C_VEL
LIN {X 0,Y 388.742,Z 554.707,A -85,B 0,C 180,E1 -11610,E2 -11610} C_VEL
LIN {X 0,Y 388.743,Z 554.488,A -85,B 0,C 180,E1 -11611.036,E2 -11611.036} C_VEL
LIN {X 0,Y 388.788,Z 553.876,A -85,B 0,C 180,E1 -11612.072,E2 -11612.072} C_VEL
LIN {X 0,Y 388.729,Z 551.452,A -85,B 0,C 180,E1 -11614.147,E2 -11614.147} C_VEL
LIN {X 0,Y 388.831,Z 548.034,A -85,B 0,C 180,E1 -11615.901,E2 -11615.901} C_VEL
LIN {X 0,Y 389.078,Z 542.867,A -85,B 0,C 180,E1 -11617.786,E2 -11617.786} C_VEL
LIN {X 0,Y 389.453,Z 537.295,A -85,B 0,C 180,E1 -11619.347,E2 -11619.347} C_VEL
LIN {X 0,Y 389.963,Z 530.344,A -85,B 0,C 180,E1 -11620.908,E2 -11620.908} C_VEL
LIN {X 0,Y 390.796,Z 521.666,A -85,B 0,C 180,E1 -11622.463,E2 -11622.463} C_VEL
LIN {X 0,Y 391.531,Z 513.09,A -85,B 0,C 180,E1 -11623.716,E2 -11623.716} C_VEL
LIN {X 0,Y 392.293,Z 503.007,A -85,B 0,C 180,E1 -11624.924,E2 -11624.924} C_VEL
LIN {X 0,Y 393.19,Z 492.344,A -85,B 0,C 180,E1 -11625.951,E2 -11625.951} C_VEL
LIN {X 0,Y 394.092,Z 481.093,A -85,B 0,C 180,E1 -11626.802,E2 -11626.802} C_VEL
LIN {X 0,Y 393.905,Z 475.967,A -85,B 0,C 180,E1 -11627.146,E2 -11627.146} C_VEL
LIN {X 0,Y 392.153,Z 462.512,A -85,B 0,C 180,E1 -11627.924,E2 -11627.924} C_VEL
LIN {X 0,Y 389.883,Z 448.784,A -85,B 0,C 180,E1 -11628.507,E2 -11628.507} C_VEL
LIN {X 0,Y 389.578,Z 446.603,A -85,B 0,C 180,E1 -11628.607,E2 -11628.607} C_VEL
LIN {X 0,Y 390.048,Z 438.263,A -85,B 0,C 180,E1 -11632.234,E2 -11632.234} C_VEL
LIN {X 0,Y 390.618,Z 429.809,A -85,B 0,C 180,E1 -11635.894,E2 -11635.894} C_VEL
LIN {X 0,Y 391.168,Z 422.64,A -85,B 0,C 180,E1 -11639.019,E2 -11639.019} C_VEL
LIN {X 0,Y 391.853,Z 414.724,A -85,B 0,C 180,E1 -11642.552,E2 -11642.552} C_VEL
LIN {X 0,Y 392.46,Z 408.231,A -85,B 0,C 180,E1 -11645.591,E2 -11645.591} C_VEL
LIN {X 0,Y 392.264,Z 404.332,A -85,B 0,C 180,E1 -11647.529,E2 -11647.529} C_VEL
LIN {X 0,Y 391.407,Z 399.148,A -85,B 0,C 180,E1 -11650.271,E2 -11650.271} C_VEL
LIN {X 0,Y 390.468,Z 394.042,A -85,B 0,C 180,E1 -11653.154,E2 -11653.154} C_VEL
LIN {X 0,Y 390.085,Z 391.904,A -85,B 0,C 180,E1 -11654.485,E2 -11654.485} C_VEL
LIN {X 0,Y 390.034,Z 391.903,A -85,B 0,C 180,E1 -11658.187,E2 -11658.187} C_VEL
LIN {X 0,Y 390.095,Z 391.896,A -85,B 0,C 180,E1 -11660.908,E2 -11660.908} C_VEL
LIN {X 0,Y 390.088,Z 391.896,A -85,B 0,C 180,E1 -11664.793,E2 -11664.793} C_VEL
LIN {X 0,Y 390.034,Z 391.898,A -85,B 0,C 180,E1 -11667.875,E2 -11667.875} C_VEL
LIN {X 0,Y 390.061,Z 391.899,A -85,B 0,C 180,E1 -11670.891,E2 -11670.891} C_VEL
LIN {X 0,Y 390.121,Z 391.889,A -85,B 0,C 180,E1 -11674.257,E2 -11674.257} C_VEL
LIN {X 0,Y 390.042,Z 391.897,A -85,B 0,C 180,E1 -11677.766,E2 -11677.766} C_VEL
LIN {X 0,Y 390.109,Z 391.89,A -85,B 0,C 180,E1 -11681.078,E2 -11681.078} C_VEL
LIN {X 0,Y 390.143,Z 391.887,A -85,B 0,C 180,E1 -11684.323,E2 -11684.323} C_VEL
LIN {X 0,Y 390.181,Z 391.879,A -85,B 0,C 180,E1 -11687.517,E2 -11687.517} C_VEL
LIN {X 0,Y 390.318,Z 391.863,A -85,B 0,C 180,E1 -11691.718,E2 -11691.718} C_VEL
LIN {X 0,Y 390.334,Z 391.861,A -85,B 0,C 180,E1 -11693.798,E2 -11693.798} C_VEL
LIN {X 0,Y 390.421,Z 391.851,A -85,B 0,C 180,E1 -11697.937,E2 -11697.937} C_VEL
LIN {X 0,Y 390.554,Z 391.836,A -85,B 0,C 180,E1 -11700,E2 -11700} C_VEL
LIN {X 0,Y 390.313,Z 391.863,A -85,B 0,C 180,E1 -11703.097,E2 -11703.097} C_VEL
LIN {X 0,Y 390.313,Z 391.864,A -85,B 0,C 180,E1 -11706.652,E2 -11706.652} C_VEL
LIN {X 0,Y 390.208,Z 391.876,A -85,B 0,C 180,E1 -11709.329,E2 -11709.329} C_VEL
LIN {X 0,Y 390.197,Z 391.878,A -85,B 0,C 180,E1 -11713.438,E2 -11713.438} C_VEL
LIN {X 0,Y 390.152,Z 391.884,A -85,B 0,C 180,E1 -11717.308,E2 -11717.308} C_VEL
LIN {X 0,Y 390.09,Z 391.893,A -85,B 0,C 180,E1 -11720.47,E2 -11720.47} C_VEL
LIN {X 0,Y 390.076,Z 391.893,A -85,B 0,C 180,E1 -11723.352,E2 -11723.352} C_VEL
LIN {X 0,Y 390.116,Z 391.888,A -85,B 0,C 180,E1 -11726.768,E2 -11726.768} C_VEL
LIN {X 0,Y 390.042,Z 391.899,A -85,B 0,C 180,E1 -11730.3,E2 -11730.3} C_VEL
LIN {X 0,Y 390.071,Z 391.898,A -85,B 0,C 180,E1 -11734.025,E2 -11734.025} C_VEL
LIN {X 0,Y 390.048,Z 391.899,A -85,B 0,C 180,E1 -11737.551,E2 -11737.551} C_VEL
LIN {X 0,Y 390.06,Z 391.895,A -85,B 0,C 180,E1 -11740.822,E2 -11740.822} C_VEL
LIN {X 0,Y 390.061,Z 391.899,A -85,B 0,C 180,E1 -11743.887,E2 -11743.887} C_VEL
LIN {X 0,Y 390.118,Z 391.887,A -85,B 0,C 180,E1 -11746.798,E2 -11746.798} C_VEL
LIN {X 0,Y 390.072,Z 391.899,A -85,B 0,C 180,E1 -11749.562,E2 -11749.562} C_VEL
LIN {X 0,Y 390.038,Z 391.897,A -85,B 0,C 180,E1 -11752.451,E2 -11752.451} C_VEL
LIN {X 0,Y 389.926,Z 391.912,A -85,B 0,C 180,E1 -11754.776,E2 -11754.776} C_VEL
LIN {X 0,Y 389.579,Z 391.959,A -85,B 0,C 180,E1 -11757.982,E2 -11757.982} C_VEL
LIN {X 0,Y 389.53,Z 391.965,A -85,B 0,C 180,E1 -11758.451,E2 -11758.451} C_VEL
LIN {X 0,Y 389.475,Z 393.888,A -85,B 0,C 180,E1 -11760.843,E2 -11760.843} C_VEL
LIN {X 0,Y 389.38,Z 397.213,A -85,B 0,C 180,E1 -11764.484,E2 -11764.484} C_VEL
LIN {X 0,Y 389.249,Z 400.35,A -85,B 0,C 180,E1 -11767.718,E2 -11767.718} C_VEL
LIN {X 0,Y 389.196,Z 403.806,A -85,B 0,C 180,E1 -11771.032,E2 -11771.032} C_VEL
LIN {X 0,Y 389.219,Z 404.31,A -85,B 0,C 180,E1 -11771.51,E2 -11771.51} C_VEL
LIN {X 0,Y 393.154,Z 418.793,A -85,B 0,C 180,E1 -11772.251,E2 -11772.251} C_VEL
LIN {X 0,Y 395.231,Z 428.918,A -85,B 0,C 180,E1 -11772.894,E2 -11772.894} C_VEL
LIN {X 0,Y 394.534,Z 440.986,A -85,B 0,C 180,E1 -11773.707,E2 -11773.707} C_VEL
LIN {X 0,Y 393.772,Z 451.57,A -85,B 0,C 180,E1 -11774.63,E2 -11774.63} C_VEL
LIN {X 0,Y 392.936,Z 461.964,A -85,B 0,C 180,E1 -11775.763,E2 -11775.763} C_VEL
LIN {X 0,Y 392.085,Z 471.535,A -85,B 0,C 180,E1 -11777.052,E2 -11777.052} C_VEL
LIN {X 0,Y 391.352,Z 479.369,A -85,B 0,C 180,E1 -11778.344,E2 -11778.344} C_VEL
LIN {X 0,Y 390.616,Z 487.023,A -85,B 0,C 180,E1 -11779.897,E2 -11779.897} C_VEL
LIN {X 0,Y 389.91,Z 494.042,A -85,B 0,C 180,E1 -11781.709,E2 -11781.709} C_VEL
LIN {X 0,Y 389.561,Z 498.479,A -85,B 0,C 180,E1 -11783.18,E2 -11783.18} C_VEL
LIN {X 0,Y 389.149,Z 502.29,A -85,B 0,C 180,E1 -11784.819,E2 -11784.819} C_VEL
LIN {X 0,Y 389.176,Z 504.126,A -85,B 0,C 180,E1 -11785.858,E2 -11785.858} C_VEL
LIN {X 0,Y 389.082,Z 505.515,A -85,B 0,C 180,E1 -11786.894,E2 -11786.894} C_VEL
LIN {X 0,Y 388.843,Z 507.118,A -85,B 0,C 180,E1 -11788.964,E2 -11788.964} C_VEL
LIN {X 0,Y 388.827,Z 507.35,A -85,B 0,C 180,E1 -11790,E2 -11790} C_VEL
LIN {X 0,Y 388.938,Z 506.578,A -85,B 0,C 180,E1 -11792.071,E2 -11792.071} C_VEL
LIN {X 0,Y 389.076,Z 505.615,A -85,B 0,C 180,E1 -11793.107,E2 -11793.107} C_VEL
LIN {X 0,Y 389.175,Z 504.269,A -85,B 0,C 180,E1 -11794.142,E2 -11794.142} C_VEL
LIN {X 0,Y 389.236,Z 501.434,A -85,B 0,C 180,E1 -11795.699,E2 -11795.699} C_VEL
LIN {X 0,Y 389.596,Z 497.571,A -85,B 0,C 180,E1 -11797.255,E2 -11797.255} C_VEL
LIN {X 0,Y 390.052,Z 492.588,A -85,B 0,C 180,E1 -11798.81,E2 -11798.81} C_VEL
LIN {X 0,Y 390.716,Z 486.305,A -85,B 0,C 180,E1 -11800.363,E2 -11800.363} C_VEL
LIN {X 0,Y 391.428,Z 478.444,A -85,B 0,C 180,E1 -11801.916,E2 -11801.916} C_VEL
LIN {X 0,Y 392.369,Z 468.653,A -85,B 0,C 180,E1 -11803.465,E2 -11803.465} C_VEL
LIN {X 0,Y 393.27,Z 459.08,A -85,B 0,C 180,E1 -11804.672,E2 -11804.672} C_VEL
LIN {X 0,Y 394.007,Z 448.181,A -85,B 0,C 180,E1 -11805.785,E2 -11805.785} C_VEL
LIN {X 0,Y 394.88,Z 435.993,A -85,B 0,C 180,E1 -11806.755,E2 -11806.755} C_VEL
LIN {X 0,Y 395.158,Z 427.882,A -85,B 0,C 180,E1 -11807.269,E2 -11807.269} C_VEL
LIN {X 0,Y 393.19,Z 418.866,A -85,B 0,C 180,E1 -11807.843,E2 -11807.843} C_VEL
LIN {X 0,Y 392.01,Z 417.039,A -85,B 0,C 180,E1 -11807.985,E2 -11807.985} C_VEL
LIN {X 0,Y 385.009,Z 413.059,A -85,B 0,C 180,E1 -11808.506,E2 -11808.506} C_VEL
LIN {X 0,Y 384.051,Z 411.471,A -85,B 0,C 180,E1 -11808.616,E2 -11808.616} C_VEL
LIN {X 0,Y 382.114,Z 404.672,A -85,B 0,C 180,E1 -11808.958,E2 -11808.958} C_VEL
LIN {X 0,Y 382.221,Z 400.853,A -85,B 0,C 180,E1 -11812.714,E2 -11812.714} C_VEL
LIN {X 0,Y 382.306,Z 397.542,A -85,B 0,C 180,E1 -11816.181,E2 -11816.181} C_VEL
LIN {X 0,Y 382.446,Z 394.324,A -85,B 0,C 180,E1 -11819.747,E2 -11819.747} C_VEL
LIN {X 0,Y 382.499,Z 393.241,A -85,B 0,C 180,E1 -11820.962,E2 -11820.962} C_VEL
LIN {X 0,Y 382.615,Z 392.827,A -85,B 0,C 180,E1 -11822.334,E2 -11822.334} C_VEL
LIN {X 0,Y 382.953,Z 392.781,A -85,B 0,C 180,E1 -11825.964,E2 -11825.964} C_VEL
LIN {X 0,Y 383.005,Z 392.778,A -85,B 0,C 180,E1 -11828.601,E2 -11828.601} C_VEL
LIN {X 0,Y 382.987,Z 392.775,A -85,B 0,C 180,E1 -11831.348,E2 -11831.348} C_VEL
LIN {X 0,Y 382.999,Z 392.779,A -85,B 0,C 180,E1 -11834.304,E2 -11834.304} C_VEL
LIN {X 0,Y 383.013,Z 392.772,A -85,B 0,C 180,E1 -11837.24,E2 -11837.24} C_VEL
LIN {X 0,Y 383.02,Z 392.777,A -85,B 0,C 180,E1 -11840.413,E2 -11840.413} C_VEL
LIN {X 0,Y 383.03,Z 392.774,A -85,B 0,C 180,E1 -11844.045,E2 -11844.045} C_VEL
LIN {X 0,Y 382.991,Z 392.776,A -85,B 0,C 180,E1 -11847.578,E2 -11847.578} C_VEL
LIN {X 0,Y 382.996,Z 392.779,A -85,B 0,C 180,E1 -11850.3,E2 -11850.3} C_VEL
LIN {X 0,Y 383.084,Z 392.769,A -85,B 0,C 180,E1 -11854.021,E2 -11854.021} C_VEL
LIN {X 0,Y 382.995,Z 392.774,A -85,B 0,C 180,E1 -11857.334,E2 -11857.334} C_VEL
LIN {X 0,Y 383.064,Z 392.766,A -85,B 0,C 180,E1 -11860.716,E2 -11860.716} C_VEL
LIN {X 0,Y 383.086,Z 392.769,A -85,B 0,C 180,E1 -11864.027,E2 -11864.027} C_VEL
LIN {X 0,Y 383.141,Z 392.757,A -85,B 0,C 180,E1 -11867.284,E2 -11867.284} C_VEL
LIN {X 0,Y 383.148,Z 392.756,A -85,B 0,C 180,E1 -11870.498,E2 -11870.498} C_VEL
LIN {X 0,Y 383.28,Z 392.744,A -85,B 0,C 180,E1 -11873.684,E2 -11873.684} C_VEL
LIN {X 0,Y 383.39,Z 392.73,A -85,B 0,C 180,E1 -11877.899,E2 -11877.899} C_VEL
LIN {X 0,Y 383.522,Z 392.712,A -85,B 0,C 180,E1 -11880,E2 -11880} C_VEL
LIN {X 0,Y 383.251,Z 392.744,A -85,B 0,C 180,E1 -11883.154,E2 -11883.154} C_VEL
LIN {X 0,Y 383.292,Z 392.738,A -85,B 0,C 180,E1 -11886.316,E2 -11886.316} C_VEL
LIN {X 0,Y 383.265,Z 392.741,A -85,B 0,C 180,E1 -11888.436,E2 -11888.436} C_VEL
LIN {X 0,Y 383.112,Z 392.765,A -85,B 0,C 180,E1 -11891.642,E2 -11891.642} C_VEL
LIN {X 0,Y 383.117,Z 392.76,A -85,B 0,C 180,E1 -11894.881,E2 -11894.881} C_VEL
LIN {X 0,Y 383.066,Z 392.766,A -85,B 0,C 180,E1 -11898.173,E2 -11898.173} C_VEL
LIN {X 0,Y 382.997,Z 392.779,A -85,B 0,C 180,E1 -11901.531,E2 -11901.531} C_VEL
LIN {X 0,Y 383.056,Z 392.77,A -85,B 0,C 180,E1 -11904.96,E2 -11904.96} C_VEL
LIN {X 0,Y 383.033,Z 392.769,A -85,B 0,C 180,E1 -11908.27,E2 -11908.27} C_VEL
LIN {X 0,Y 383.013,Z 392.772,A -85,B 0,C 180,E1 -11912.149,E2 -11912.149} C_VEL
LIN {X 0,Y 383.021,Z 392.773,A -85,B 0,C 180,E1 -11914.668,E2 -11914.668} C_VEL
LIN {X 0,Y 383.003,Z 392.774,A -85,B 0,C 180,E1 -11917.904,E2 -11917.904} C_VEL
LIN {X 0,Y 382.987,Z 392.781,A -85,B 0,C 180,E1 -11921.347,E2 -11921.347} C_VEL
LIN {X 0,Y 383.029,Z 392.776,A -85,B 0,C 180,E1 -11924.948,E2 -11924.948} C_VEL
LIN {X 0,Y 383.053,Z 393.007,A -85,B 0,C 180,E1 -11925.315,E2 -11925.315} C_VEL
LIN {X 0,Y 384.081,Z 398.576,A -85,B 0,C 180,E1 -11928.61,E2 -11928.61} C_VEL
LIN {X 0,Y 385.101,Z 404.215,A -85,B 0,C 180,E1 -11931.697,E2 -11931.697} C_VEL
LIN {X 0,Y 385.48,Z 407.384,A -85,B 0,C 180,E1 -11933.341,E2 -11933.341} C_VEL
LIN {X 0,Y 385.213,Z 411.942,A -85,B 0,C 180,E1 -11935.557,E2 -11935.557} C_VEL
LIN {X 0,Y 384.609,Z 418.46,A -85,B 0,C 180,E1 -11938.615,E2 -11938.615} C_VEL
LIN {X 0,Y 383.927,Z 426.29,A -85,B 0,C 180,E1 -11942.173,E2 -11942.173} C_VEL
LIN {X 0,Y 383.291,Z 434.057,A -85,B 0,C 180,E1 -11945.634,E2 -11945.634} C_VEL
LIN {X 0,Y 382.736,Z 442.957,A -85,B 0,C 180,E1 -11949.58,E2 -11949.58} C_VEL
LIN {X 0,Y 382.517,Z 446.321,A -85,B 0,C 180,E1 -11951.071,E2 -11951.071} C_VEL
LIN {X 0,Y 384.843,Z 460.218,A -85,B 0,C 180,E1 -11951.638,E2 -11951.638} C_VEL
LIN {X 0,Y 386.462,Z 472.374,A -85,B 0,C 180,E1 -11952.322,E2 -11952.322} C_VEL
LIN {X 0,Y 387.28,Z 480.859,A -85,B 0,C 180,E1 -11952.904,E2 -11952.904} C_VEL
LIN {X 0,Y 386.378,Z 491.933,A -85,B 0,C 180,E1 -11953.76,E2 -11953.76} C_VEL
LIN {X 0,Y 385.299,Z 503.772,A -85,B 0,C 180,E1 -11954.934,E2 -11954.934} C_VEL
LIN {X 0,Y 384.447,Z 514.307,A -85,B 0,C 180,E1 -11956.252,E2 -11956.252} C_VEL
LIN {X 0,Y 383.652,Z 522.835,A -85,B 0,C 180,E1 -11957.57,E2 -11957.57} C_VEL
LIN {X 0,Y 382.841,Z 531.161,A -85,B 0,C 180,E1 -11959.154,E2 -11959.154} C_VEL
LIN {X 0,Y 382.334,Z 537.885,A -85,B 0,C 180,E1 -11960.744,E2 -11960.744} C_VEL
LIN {X 0,Y 381.954,Z 544.048,A -85,B 0,C 180,E1 -11962.6,E2 -11962.6} C_VEL
LIN {X 0,Y 381.735,Z 547.957,A -85,B 0,C 180,E1 -11964.143,E2 -11964.143} C_VEL
LIN {X 0,Y 381.658,Z 551.018,A -85,B 0,C 180,E1 -11965.776,E2 -11965.776} C_VEL
LIN {X 0,Y 381.704,Z 553.444,A -85,B 0,C 180,E1 -11967.89,E2 -11967.89} C_VEL
LIN {X 0,Y 381.676,Z 554.057,A -85,B 0,C 180,E1 -11968.945,E2 -11968.945} C_VEL
LIN {X 0,Y 381.672,Z 554.276,A -85,B 0,C 180,E1 -11970,E2 -11970} C_VEL
LIN {X 0,Y 381.676,Z 554.057,A -85,B 0,C 180,E1 -11971.055,E2 -11971.055} C_VEL
LIN {X 0,Y 381.704,Z 553.444,A -85,B 0,C 180,E1 -11972.11,E2 -11972.11} C_VEL
LIN {X 0,Y 381.658,Z 551.02,A -85,B 0,C 180,E1 -11974.224,E2 -11974.224} C_VEL
LIN {X 0,Y 381.732,Z 547.965,A -85,B 0,C 180,E1 -11975.852,E2 -11975.852} C_VEL
LIN {X 0,Y 381.928,Z 544.04,A -85,B 0,C 180,E1 -11977.401,E2 -11977.401} C_VEL
LIN {X 0,Y 382.334,Z 537.879,A -85,B 0,C 180,E1 -11979.256,E2 -11979.256} C_VEL
LIN {X 0,Y 382.84,Z 531.152,A -85,B 0,C 180,E1 -11980.846,E2 -11980.846} C_VEL
LIN {X 0,Y 383.648,Z 522.823,A -85,B 0,C 180,E1 -11982.43,E2 -11982.43} C_VEL
LIN {X 0,Y 384.441,Z 514.29,A -85,B 0,C 180,E1 -11983.748,E2 -11983.748} C_VEL
LIN {X 0,Y 385.292,Z 503.75,A -85,B 0,C 180,E1 -11985.066,E2 -11985.066} C_VEL
LIN {X 0,Y 386.357,Z 491.907,A -85,B 0,C 180,E1 -11986.241,E2 -11986.241} C_VEL
LIN {X 0,Y 387.267,Z 480.817,A -85,B 0,C 180,E1 -11987.096,E2 -11987.096} C_VEL
LIN {X 0,Y 386.212,Z 470.446,A -85,B 0,C 180,E1 -11987.798,E2 -11987.798} C_VEL
LIN {X 0,Y 384.442,Z 457.807,A -85,B 0,C 180,E1 -11988.47,E2 -11988.47} C_VEL
LIN {X 0,Y 382.531,Z 446.254,A -85,B 0,C 180,E1 -11988.928,E2 -11988.928} C_VEL
LIN {X 0,Y 383.044,Z 437.879,A -85,B 0,C 180,E1 -11992.663,E2 -11992.663} C_VEL
LIN {X 0,Y 383.702,Z 428.876,A -85,B 0,C 180,E1 -11996.663,E2 -11996.663} C_VEL
LIN {X 0,Y 384.228,Z 422.319,A -85,B 0,C 180,E1 -11999.595,E2 -11999.595} C_VEL
LIN {X 0,Y 384.882,Z 415.17,A -85,B 0,C 180,E1 -12002.863,E2 -12002.863} C_VEL
LIN {X 0,Y 385.459,Z 409.255,A -85,B 0,C 180,E1 -12005.694,E2 -12005.694} C_VEL
LIN {X 0,Y 385.279,Z 405.417,A -85,B 0,C 180,E1 -12007.644,E2 -12007.644} C_VEL
LIN {X 0,Y 384.142,Z 398.938,A -85,B 0,C 180,E1 -12011.196,E2 -12011.196} C_VEL
LIN {X 0,Y 383.086,Z 392.981,A -85,B 0,C 180,E1 -12014.69,E2 -12014.69} C_VEL
LIN {X 0,Y 383.012,Z 392.778,A -85,B 0,C 180,E1 -12017.24,E2 -12017.24} C_VEL
LIN {X 0,Y 383.019,Z 392.778,A -85,B 0,C 180,E1 -12020.413,E2 -12020.413} C_VEL
LIN {X 0,Y 383.029,Z 392.77,A -85,B 0,C 180,E1 -12024.045,E2 -12024.045} C_VEL
LIN {X 0,Y 382.989,Z 392.775,A -85,B 0,C 180,E1 -12027.578,E2 -12027.578} C_VEL
LIN {X 0,Y 382.995,Z 392.776,A -85,B 0,C 180,E1 -12030.3,E2 -12030.3} C_VEL
LIN {X 0,Y 383.083,Z 392.764,A -85,B 0,C 180,E1 -12034.021,E2 -12034.021} C_VEL
LIN {X 0,Y 383.011,Z 392.773,A -85,B 0,C 180,E1 -12037.335,E2 -12037.335} C_VEL
LIN {X 0,Y 383.064,Z 392.772,A -85,B 0,C 180,E1 -12040.716,E2 -12040.716} C_VEL
LIN {X 0,Y 383.084,Z 392.764,A -85,B 0,C 180,E1 -12044.027,E2 -12044.027} C_VEL
LIN {X 0,Y 383.145,Z 392.756,A -85,B 0,C 180,E1 -12047.284,E2 -12047.284} C_VEL
LIN {X 0,Y 383.16,Z 392.76,A -85,B 0,C 180,E1 -12050.498,E2 -12050.498} C_VEL
LIN {X 0,Y 383.277,Z 392.744,A -85,B 0,C 180,E1 -12052.625,E2 -12052.625} C_VEL
LIN {X 0,Y 383.202,Z 392.752,A -85,B 0,C 180,E1 -12054.739,E2 -12054.739} C_VEL
LIN {X 0,Y 383.389,Z 392.727,A -85,B 0,C 180,E1 -12057.899,E2 -12057.899} C_VEL
LIN {X 0,Y 383.523,Z 392.711,A -85,B 0,C 180,E1 -12060,E2 -12060} C_VEL
LIN {X 0,Y 383.249,Z 392.743,A -85,B 0,C 180,E1 -12063.154,E2 -12063.154} C_VEL
LIN {X 0,Y 383.272,Z 392.742,A -85,B 0,C 180,E1 -12066.646,E2 -12066.646} C_VEL
LIN {X 0,Y 383.263,Z 392.745,A -85,B 0,C 180,E1 -12068.436,E2 -12068.436} C_VEL
LIN {X 0,Y 383.1,Z 392.762,A -85,B 0,C 180,E1 -12071.642,E2 -12071.642} C_VEL
LIN {X 0,Y 383.113,Z 392.76,A -85,B 0,C 180,E1 -12074.882,E2 -12074.882} C_VEL
LIN {X 0,Y 383.092,Z 392.768,A -85,B 0,C 180,E1 -12078.172,E2 -12078.172} C_VEL
LIN {X 0,Y 382.995,Z 392.776,A -85,B 0,C 180,E1 -12081.531,E2 -12081.531} C_VEL
LIN {X 0,Y 383.053,Z 392.767,A -85,B 0,C 180,E1 -12084.96,E2 -12084.96} C_VEL
LIN {X 0,Y 383.032,Z 392.773,A -85,B 0,C 180,E1 -12088.27,E2 -12088.27} C_VEL
LIN {X 0,Y 383.012,Z 392.776,A -85,B 0,C 180,E1 -12092.15,E2 -12092.15} C_VEL
LIN {X 0,Y 383.021,Z 392.771,A -85,B 0,C 180,E1 -12094.668,E2 -12094.668} C_VEL
LIN {X 0,Y 383.004,Z 392.778,A -85,B 0,C 180,E1 -12097.904,E2 -12097.904} C_VEL
LIN {X 0,Y 382.987,Z 392.778,A -85,B 0,C 180,E1 -12101.347,E2 -12101.347} C_VEL
LIN {X 0,Y 383.01,Z 392.774,A -85,B 0,C 180,E1 -12104.305,E2 -12104.305} C_VEL
LIN {X 0,Y 383.077,Z 392.766,A -85,B 0,C 180,E1 -12107.249,E2 -12107.249} C_VEL
LIN {X 0,Y 383.02,Z 392.771,A -85,B 0,C 180,E1 -12110.413,E2 -12110.413} C_VEL
LIN {X 0,Y 382.952,Z 392.782,A -85,B 0,C 180,E1 -12114.036,E2 -12114.036} C_VEL
LIN {X 0,Y 382.688,Z 392.82,A -85,B 0,C 180,E1 -12116.568,E2 -12116.568} C_VEL
LIN {X 0,Y 382.457,Z 393.146,A -85,B 0,C 180,E1 -12119.034,E2 -12119.034} C_VEL
LIN {X 0,Y 382.332,Z 396.353,A -85,B 0,C 180,E1 -12122.642,E2 -12122.642} C_VEL
LIN {X 0,Y 382.282,Z 398.524,A -85,B 0,C 180,E1 -12124.986,E2 -12124.986} C_VEL
LIN {X 0,Y 382.168,Z 401.868,A -85,B 0,C 180,E1 -12128.42,E2 -12128.42} C_VEL
LIN {X 0,Y 382.169,Z 404.732,A -85,B 0,C 180,E1 -12131.159,E2 -12131.159} C_VEL
LIN {X 0,Y 386.122,Z 419.133,A -85,B 0,C 180,E1 -12131.911,E2 -12131.911} C_VEL
LIN {X 0,Y 388.431,Z 429.889,A -85,B 0,C 180,E1 -12132.617,E2 -12132.617} C_VEL
LIN {X 0,Y 387.745,Z 441.42,A -85,B 0,C 180,E1 -12133.413,E2 -12133.413} C_VEL
LIN {X 0,Y 386.932,Z 452.212,A -85,B 0,C 180,E1 -12134.373,E2 -12134.373} C_VEL
LIN {X 0,Y 386.071,Z 462.4,A -85,B 0,C 180,E1 -12135.505,E2 -12135.505} C_VEL
LIN {X 0,Y 385.192,Z 471.969,A -85,B 0,C 180,E1 -12136.817,E2 -12136.817} C_VEL
LIN {X 0,Y 384.412,Z 479.804,A -85,B 0,C 180,E1 -12138.131,E2 -12138.131} C_VEL
LIN {X 0,Y 383.654,Z 487.455,A -85,B 0,C 180,E1 -12139.711,E2 -12139.711} C_VEL
LIN {X 0,Y 382.913,Z 494.474,A -85,B 0,C 180,E1 -12141.557,E2 -12141.557} C_VEL
LIN {X 0,Y 382.496,Z 499.204,A -85,B 0,C 180,E1 -12143.164,E2 -12143.164} C_VEL
LIN {X 0,Y 382.093,Z 502.722,A -85,B 0,C 180,E1 -12144.723,E2 -12144.723} C_VEL
LIN {X 0,Y 382.092,Z 504.559,A -85,B 0,C 180,E1 -12145.781,E2 -12145.781} C_VEL
LIN {X 0,Y 382.025,Z 505.946,A -85,B 0,C 180,E1 -12146.836,E2 -12146.836} C_VEL
LIN {X 0,Y 381.772,Z 507.549,A -85,B 0,C 180,E1 -12148.945,E2 -12148.945} C_VEL
LIN {X 0,Y 381.752,Z 507.781,A -85,B 0,C 180,E1 -12150,E2 -12150} C_VEL
LIN {X 0,Y 381.873,Z 507.009,A -85,B 0,C 180,E1 -12152.11,E2 -12152.11} C_VEL
LIN {X 0,Y 382.02,Z 506.045,A -85,B 0,C 180,E1 -12153.164,E2 -12153.164} C_VEL
LIN {X 0,Y 382.091,Z 504.701,A -85,B 0,C 180,E1 -12154.219,E2 -12154.219} C_VEL
LIN {X 0,Y 382.2,Z 501.863,A -85,B 0,C 180,E1 -12155.805,E2 -12155.805} C_VEL
LIN {X 0,Y 382.564,Z 498.002,A -85,B 0,C 180,E1 -12157.389,E2 -12157.389} C_VEL
LIN {X 0,Y 383.042,Z 493.018,A -85,B 0,C 180,E1 -12158.972,E2 -12158.972} C_VEL
LIN {X 0,Y 383.732,Z 486.736,A -85,B 0,C 180,E1 -12160.553,E2 -12160.553} C_VEL
LIN {X 0,Y 384.508,Z 478.872,A -85,B 0,C 180,E1 -12162.134,E2 -12162.134} C_VEL
LIN {X 0,Y 385.49,Z 469.081,A -85,B 0,C 180,E1 -12163.71,E2 -12163.71} C_VEL
LIN {X 0,Y 386.421,Z 459.629,A -85,B 0,C 180,E1 -12164.924,E2 -12164.924} C_VEL
LIN {X 0,Y 387.199,Z 448.607,A -85,B 0,C 180,E1 -12166.07,E2 -12166.07} C_VEL
LIN {X 0,Y 388.089,Z 436.557,A -85,B 0,C 180,E1 -12167.047,E2 -12167.047} C_VEL
LIN {X 0,Y 388.337,Z 428.907,A -85,B 0,C 180,E1 -12167.546,E2 -12167.546} C_VEL
LIN {X 0,Y 385.405,Z 416.187,A -85,B 0,C 180,E1 -12168.359,E2 -12168.359} C_VEL
LIN {X 0,Y 384.051,Z 411.471,A -85,B 0,C 180,E1 -12168.616,E2 -12168.616} C_VEL
LIN {X 0,Y 382.89,Z 408.455,A -85,B 0,C 180,E1 -12168.89,E2 -12168.89} C_VEL
LIN {X 0,Y 381.464,Z 406.242,A -85,B 0,C 180,E1 -12169.295,E2 -12169.295} C_VEL
LIN {X 0,Y 379.233,Z 404.124,A -85,B 0,C 180,E1 -12170.047,E2 -12170.047} C_VEL
LIN {X 0,Y 376.111,Z 402.714,A -85,B 0,C 180,E1 -12171.556,E2 -12171.556} C_VEL
LIN {X 0,Y 375.214,Z 401.878,A -85,B 0,C 180,E1 -12172.52,E2 -12172.52} C_VEL
LIN {X 0,Y 375.171,Z 401.562,A -85,B 0,C 180,E1 -12172.845,E2 -12172.845} C_VEL
LIN {X 0,Y 375.263,Z 398.588,A -85,B 0,C 180,E1 -12175.978,E2 -12175.978} C_VEL
LIN {X 0,Y 375.365,Z 395.728,A -85,B 0,C 180,E1 -12179.131,E2 -12179.131} C_VEL
LIN {X 0,Y 375.476,Z 393.717,A -85,B 0,C 180,E1 -12181.608,E2 -12181.608} C_VEL
LIN {X 0,Y 375.845,Z 393.665,A -85,B 0,C 180,E1 -12185.428,E2 -12185.428} C_VEL
LIN {X 0,Y 375.974,Z 393.653,A -85,B 0,C 180,E1 -12188.27,E2 -12188.27} C_VEL
LIN {X 0,Y 375.937,Z 393.653,A -85,B 0,C 180,E1 -12191.601,E2 -12191.601} C_VEL
LIN {X 0,Y 375.93,Z 393.654,A -85,B 0,C 180,E1 -12195.269,E2 -12195.269} C_VEL
LIN {X 0,Y 375.938,Z 393.659,A -85,B 0,C 180,E1 -12198.399,E2 -12198.399} C_VEL
LIN {X 0,Y 375.98,Z 393.649,A -85,B 0,C 180,E1 -12201.729,E2 -12201.729} C_VEL
LIN {X 0,Y 375.984,Z 393.647,A -85,B 0,C 180,E1 -12205.333,E2 -12205.333} C_VEL
LIN {X 0,Y 375.962,Z 393.654,A -85,B 0,C 180,E1 -12208.438,E2 -12208.438} C_VEL
LIN {X 0,Y 375.988,Z 393.653,A -85,B 0,C 180,E1 -12212.14,E2 -12212.14} C_VEL
LIN {X 0,Y 376.009,Z 393.646,A -85,B 0,C 180,E1 -12214.539,E2 -12214.539} C_VEL
LIN {X 0,Y 375.961,Z 393.657,A -85,B 0,C 180,E1 -12218.045,E2 -12218.045} C_VEL
LIN {X 0,Y 376.028,Z 393.644,A -85,B 0,C 180,E1 -12221.474,E2 -12221.474} C_VEL
LIN {X 0,Y 376.063,Z 393.638,A -85,B 0,C 180,E1 -12224.833,E2 -12224.833} C_VEL
LIN {X 0,Y 376.054,Z 393.642,A -85,B 0,C 180,E1 -12228.137,E2 -12228.137} C_VEL
LIN {X 0,Y 376.205,Z 393.625,A -85,B 0,C 180,E1 -12231.938,E2 -12231.938} C_VEL
LIN {X 0,Y 376.173,Z 393.624,A -85,B 0,C 180,E1 -12234.64,E2 -12234.64} C_VEL
LIN {X 0,Y 376.356,Z 393.606,A -85,B 0,C 180,E1 -12237.86,E2 -12237.86} C_VEL
LIN {X 0,Y 376.492,Z 393.587,A -85,B 0,C 180,E1 -12240,E2 -12240} C_VEL
LIN {X 0,Y 376.189,Z 393.624,A -85,B 0,C 180,E1 -12243.213,E2 -12243.213} C_VEL
LIN {X 0,Y 376.252,Z 393.614,A -85,B 0,C 180,E1 -12246.435,E2 -12246.435} C_VEL
LIN {X 0,Y 376.211,Z 393.619,A -85,B 0,C 180,E1 -12248.595,E2 -12248.595} C_VEL
LIN {X 0,Y 376.064,Z 393.64,A -85,B 0,C 180,E1 -12251.863,E2 -12251.863} C_VEL
LIN {X 0,Y 376.064,Z 393.641,A -85,B 0,C 180,E1 -12255.167,E2 -12255.167} C_VEL
LIN {X 0,Y 376.012,Z 393.644,A -85,B 0,C 180,E1 -12258.527,E2 -12258.527} C_VEL
LIN {X 0,Y 375.967,Z 393.651,A -85,B 0,C 180,E1 -12261.954,E2 -12261.954} C_VEL
LIN {X 0,Y 376.01,Z 393.649,A -85,B 0,C 180,E1 -12265.461,E2 -12265.461} C_VEL
LIN {X 0,Y 375.965,Z 393.654,A -85,B 0,C 180,E1 -12269.08,E2 -12269.08} C_VEL
LIN {X 0,Y 375.952,Z 393.654,A -85,B 0,C 180,E1 -12272.828,E2 -12272.828} C_VEL
LIN {X 0,Y 375.961,Z 393.654,A -85,B 0,C 180,E1 -12275.415,E2 -12275.415} C_VEL
LIN {X 0,Y 375.978,Z 393.648,A -85,B 0,C 180,E1 -12278.27,E2 -12278.27} C_VEL
LIN {X 0,Y 375.938,Z 393.66,A -85,B 0,C 180,E1 -12281.601,E2 -12281.601} C_VEL
LIN {X 0,Y 376.001,Z 393.732,A -85,B 0,C 180,E1 -12284.798,E2 -12284.798} C_VEL
LIN {X 0,Y 377.037,Z 399.364,A -85,B 0,C 180,E1 -12288.211,E2 -12288.211} C_VEL
LIN {X 0,Y 378.013,Z 404.907,A -85,B 0,C 180,E1 -12291.34,E2 -12291.34} C_VEL
LIN {X 0,Y 378.487,Z 409.068,A -85,B 0,C 180,E1 -12293.544,E2 -12293.544} C_VEL
LIN {X 0,Y 378.089,Z 414.262,A -85,B 0,C 180,E1 -12296.106,E2 -12296.106} C_VEL
LIN {X 0,Y 377.493,Z 420.154,A -85,B 0,C 180,E1 -12298.916,E2 -12298.916} C_VEL
LIN {X 0,Y 376.873,Z 427.254,A -85,B 0,C 180,E1 -12302.211,E2 -12302.211} C_VEL
LIN {X 0,Y 376.118,Z 436.189,A -85,B 0,C 180,E1 -12306.291,E2 -12306.291} C_VEL
LIN {X 0,Y 375.606,Z 443.912,A -85,B 0,C 180,E1 -12309.799,E2 -12309.799} C_VEL
LIN {X 0,Y 375.479,Z 445.9,A -85,B 0,C 180,E1 -12310.702,E2 -12310.702} C_VEL
LIN {X 0,Y 377.859,Z 459.778,A -85,B 0,C 180,E1 -12311.286,E2 -12311.286} C_VEL
LIN {X 0,Y 379.571,Z 472.905,A -85,B 0,C 180,E1 -12312.05,E2 -12312.05} C_VEL
LIN {X 0,Y 380.404,Z 480.582,A -85,B 0,C 180,E1 -12312.596,E2 -12312.596} C_VEL
LIN {X 0,Y 379.408,Z 492.936,A -85,B 0,C 180,E1 -12313.591,E2 -12313.591} C_VEL
LIN {X 0,Y 378.292,Z 504.521,A -85,B 0,C 180,E1 -12314.786,E2 -12314.786} C_VEL
LIN {X 0,Y 377.528,Z 513.875,A -85,B 0,C 180,E1 -12315.995,E2 -12315.995} C_VEL
LIN {X 0,Y 376.701,Z 522.404,A -85,B 0,C 180,E1 -12317.337,E2 -12317.337} C_VEL
LIN {X 0,Y 375.831,Z 530.728,A -85,B 0,C 180,E1 -12318.949,E2 -12318.949} C_VEL
LIN {X 0,Y 375.286,Z 537.452,A -85,B 0,C 180,E1 -12320.569,E2 -12320.569} C_VEL
LIN {X 0,Y 374.88,Z 543.614,A -85,B 0,C 180,E1 -12322.459,E2 -12322.459} C_VEL
LIN {X 0,Y 374.701,Z 546.916,A -85,B 0,C 180,E1 -12323.766,E2 -12323.766} C_VEL
LIN {X 0,Y 374.589,Z 550.587,A -85,B 0,C 180,E1 -12325.696,E2 -12325.696} C_VEL
LIN {X 0,Y 374.622,Z 553.012,A -85,B 0,C 180,E1 -12327.85,E2 -12327.85} C_VEL
LIN {X 0,Y 374.61,Z 553.627,A -85,B 0,C 180,E1 -12328.925,E2 -12328.925} C_VEL
LIN {X 0,Y 374.604,Z 553.846,A -85,B 0,C 180,E1 -12330,E2 -12330} C_VEL
LIN {X 0,Y 374.61,Z 553.627,A -85,B 0,C 180,E1 -12331.075,E2 -12331.075} C_VEL
LIN {X 0,Y 374.622,Z 553.012,A -85,B 0,C 180,E1 -12332.15,E2 -12332.15} C_VEL
LIN {X 0,Y 374.588,Z 550.587,A -85,B 0,C 180,E1 -12334.304,E2 -12334.304} C_VEL
LIN {X 0,Y 374.699,Z 546.915,A -85,B 0,C 180,E1 -12336.232,E2 -12336.232} C_VEL
LIN {X 0,Y 374.944,Z 541.996,A -85,B 0,C 180,E1 -12338.081,E2 -12338.081} C_VEL
LIN {X 0,Y 375.396,Z 536.424,A -85,B 0,C 180,E1 -12339.7,E2 -12339.7} C_VEL
LIN {X 0,Y 375.956,Z 529.471,A -85,B 0,C 180,E1 -12341.32,E2 -12341.32} C_VEL
LIN {X 0,Y 376.862,Z 520.792,A -85,B 0,C 180,E1 -12342.931,E2 -12342.931} C_VEL
LIN {X 0,Y 377.769,Z 511.356,A -85,B 0,C 180,E1 -12344.346,E2 -12344.346} C_VEL
LIN {X 0,Y 378.645,Z 500.949,A -85,B 0,C 180,E1 -12345.613,E2 -12345.613} C_VEL
LIN {X 0,Y 379.624,Z 489.92,A -85,B 0,C 180,E1 -12346.676,E2 -12346.676} C_VEL
LIN {X 0,Y 380.39,Z 480.537,A -85,B 0,C 180,E1 -12347.404,E2 -12347.404} C_VEL
LIN {X 0,Y 378.879,Z 466.998,A -85,B 0,C 180,E1 -12348.313,E2 -12348.313} C_VEL
LIN {X 0,Y 376.873,Z 453.72,A -85,B 0,C 180,E1 -12348.992,E2 -12348.992} C_VEL
LIN {X 0,Y 375.497,Z 445.826,A -85,B 0,C 180,E1 -12349.297,E2 -12349.297} C_VEL
LIN {X 0,Y 375.949,Z 438.77,A -85,B 0,C 180,E1 -12352.534,E2 -12352.534} C_VEL
LIN {X 0,Y 376.63,Z 429.81,A -85,B 0,C 180,E1 -12356.606,E2 -12356.606} C_VEL
LIN {X 0,Y 377.189,Z 423.299,A -85,B 0,C 180,E1 -12359.588,E2 -12359.588} C_VEL
LIN {X 0,Y 377.812,Z 416.769,A -85,B 0,C 180,E1 -12362.647,E2 -12362.647} C_VEL
LIN {X 0,Y 378.463,Z 410.261,A -85,B 0,C 180,E1 -12365.799,E2 -12365.799} C_VEL
LIN {X 0,Y 378.263,Z 406.388,A -85,B 0,C 180,E1 -12367.816,E2 -12367.816} C_VEL
LIN {X 0,Y 377.372,Z 401.257,A -85,B 0,C 180,E1 -12370.679,E2 -12370.679} C_VEL
LIN {X 0,Y 376.425,Z 396.152,A -85,B 0,C 180,E1 -12373.694,E2 -12373.694} C_VEL
LIN {X 0,Y 375.988,Z 393.66,A -85,B 0,C 180,E1 -12375.259,E2 -12375.259} C_VEL
LIN {X 0,Y 375.943,Z 393.658,A -85,B 0,C 180,E1 -12379.133,E2 -12379.133} C_VEL
LIN {X 0,Y 375.969,Z 393.649,A -85,B 0,C 180,E1 -12381.912,E2 -12381.912} C_VEL
LIN {X 0,Y 375.982,Z 393.65,A -85,B 0,C 180,E1 -12385.333,E2 -12385.333} C_VEL
LIN {X 0,Y 375.96,Z 393.653,A -85,B 0,C 180,E1 -12388.438,E2 -12388.438} C_VEL
LIN {X 0,Y 375.985,Z 393.648,A -85,B 0,C 180,E1 -12392.14,E2 -12392.14} C_VEL
LIN {X 0,Y 376.009,Z 393.649,A -85,B 0,C 180,E1 -12394.539,E2 -12394.539} C_VEL
LIN {X 0,Y 375.966,Z 393.651,A -85,B 0,C 180,E1 -12398.046,E2 -12398.046} C_VEL
LIN {X 0,Y 376.012,Z 393.644,A -85,B 0,C 180,E1 -12401.473,E2 -12401.473} C_VEL
LIN {X 0,Y 376.063,Z 393.641,A -85,B 0,C 180,E1 -12404.833,E2 -12404.833} C_VEL
LIN {X 0,Y 376.062,Z 393.64,A -85,B 0,C 180,E1 -12408.137,E2 -12408.137} C_VEL
LIN {X 0,Y 376.261,Z 393.614,A -85,B 0,C 180,E1 -12411.877,E2 -12411.877} C_VEL
LIN {X 0,Y 376.174,Z 393.628,A -85,B 0,C 180,E1 -12414.64,E2 -12414.64} C_VEL
LIN {X 0,Y 376.355,Z 393.603,A -85,B 0,C 180,E1 -12417.86,E2 -12417.86} C_VEL
LIN {X 0,Y 376.492,Z 393.587,A -85,B 0,C 180,E1 -12420,E2 -12420} C_VEL
LIN {X 0,Y 376.187,Z 393.622,A -85,B 0,C 180,E1 -12423.213,E2 -12423.213} C_VEL
LIN {X 0,Y 376.237,Z 393.618,A -85,B 0,C 180,E1 -12426.638,E2 -12426.638} C_VEL
LIN {X 0,Y 376.208,Z 393.622,A -85,B 0,C 180,E1 -12428.595,E2 -12428.595} C_VEL
LIN {X 0,Y 376.053,Z 393.642,A -85,B 0,C 180,E1 -12431.863,E2 -12431.863} C_VEL
LIN {X 0,Y 376.062,Z 393.638,A -85,B 0,C 180,E1 -12435.167,E2 -12435.167} C_VEL
LIN {X 0,Y 376.026,Z 393.644,A -85,B 0,C 180,E1 -12438.526,E2 -12438.526} C_VEL
LIN {X 0,Y 375.961,Z 393.656,A -85,B 0,C 180,E1 -12441.955,E2 -12441.955} C_VEL
LIN {X 0,Y 376.008,Z 393.646,A -85,B 0,C 180,E1 -12445.461,E2 -12445.461} C_VEL
LIN {X 0,Y 375.964,Z 393.65,A -85,B 0,C 180,E1 -12449.08,E2 -12449.08} C_VEL
LIN {X 0,Y 375.953,Z 393.651,A -85,B 0,C 180,E1 -12452.828,E2 -12452.828} C_VEL
LIN {X 0,Y 375.961,Z 393.653,A -85,B 0,C 180,E1 -12455.415,E2 -12455.415} C_VEL
LIN {X 0,Y 375.979,Z 393.65,A -85,B 0,C 180,E1 -12458.271,E2 -12458.271} C_VEL
LIN {X 0,Y 375.937,Z 393.658,A -85,B 0,C 180,E1 -12461.601,E2 -12461.601} C_VEL
LIN {X 0,Y 375.982,Z 393.65,A -85,B 0,C 180,E1 -12465.26,E2 -12465.26} C_VEL
LIN {X 0,Y 375.99,Z 393.647,A -85,B 0,C 180,E1 -12468.39,E2 -12468.39} C_VEL
LIN {X 0,Y 375.963,Z 393.653,A -85,B 0,C 180,E1 -12471.911,E2 -12471.911} C_VEL
LIN {X 0,Y 375.844,Z 393.665,A -85,B 0,C 180,E1 -12474.572,E2 -12474.572} C_VEL
LIN {X 0,Y 375.558,Z 393.707,A -85,B 0,C 180,E1 -12477.364,E2 -12477.364} C_VEL
LIN {X 0,Y 375.433,Z 393.72,A -85,B 0,C 180,E1 -12478.389,E2 -12478.389} C_VEL
LIN {X 0,Y 375.363,Z 395.639,A -85,B 0,C 180,E1 -12480.869,E2 -12480.869} C_VEL
LIN {X 0,Y 375.265,Z 398.903,A -85,B 0,C 180,E1 -12484.485,E2 -12484.485} C_VEL
LIN {X 0,Y 375.14,Z 402.273,A -85,B 0,C 180,E1 -12487.995,E2 -12487.995} C_VEL
LIN {X 0,Y 375.112,Z 405.174,A -85,B 0,C 180,E1 -12490.79,E2 -12490.79} C_VEL
LIN {X 0,Y 379.1,Z 419.51,A -85,B 0,C 180,E1 -12491.56,E2 -12491.56} C_VEL
LIN {X 0,Y 381.631,Z 430.838,A -85,B 0,C 180,E1 -12492.329,E2 -12492.329} C_VEL
LIN {X 0,Y 380.983,Z 441.856,A -85,B 0,C 180,E1 -12493.11,E2 -12493.11} C_VEL
LIN {X 0,Y 380.105,Z 452.869,A -85,B 0,C 180,E1 -12494.109,E2 -12494.109} C_VEL
LIN {X 0,Y 379.234,Z 462.834,A -85,B 0,C 180,E1 -12495.237,E2 -12495.237} C_VEL
LIN {X 0,Y 378.298,Z 472.404,A -85,B 0,C 180,E1 -12496.572,E2 -12496.572} C_VEL
LIN {X 0,Y 377.486,Z 480.238,A -85,B 0,C 180,E1 -12497.91,E2 -12497.91} C_VEL
LIN {X 0,Y 376.693,Z 487.889,A -85,B 0,C 180,E1 -12499.519,E2 -12499.519} C_VEL
LIN {X 0,Y 375.899,Z 494.908,A -85,B 0,C 180,E1 -12501.398,E2 -12501.398} C_VEL
LIN {X 0,Y 375.432,Z 499.927,A -85,B 0,C 180,E1 -12503.146,E2 -12503.146} C_VEL
LIN {X 0,Y 375.043,Z 503.155,A -85,B 0,C 180,E1 -12504.624,E2 -12504.624} C_VEL
LIN {X 0,Y 375.011,Z 504.992,A -85,B 0,C 180,E1 -12505.701,E2 -12505.701} C_VEL
LIN {X 0,Y 374.969,Z 506.376,A -85,B 0,C 180,E1 -12506.777,E2 -12506.777} C_VEL
LIN {X 0,Y 374.703,Z 507.98,A -85,B 0,C 180,E1 -12508.925,E2 -12508.925} C_VEL
LIN {X 0,Y 374.68,Z 508.212,A -85,B 0,C 180,E1 -12510,E2 -12510} C_VEL
LIN {X 0,Y 374.811,Z 507.439,A -85,B 0,C 180,E1 -12512.149,E2 -12512.149} C_VEL
LIN {X 0,Y 374.964,Z 506.474,A -85,B 0,C 180,E1 -12513.224,E2 -12513.224} C_VEL
LIN {X 0,Y 375.01,Z 505.133,A -85,B 0,C 180,E1 -12514.299,E2 -12514.299} C_VEL
LIN {X 0,Y 375.167,Z 502.293,A -85,B 0,C 180,E1 -12515.914,E2 -12515.914} C_VEL
LIN {X 0,Y 375.551,Z 498.431,A -85,B 0,C 180,E1 -12517.527,E2 -12517.527} C_VEL
LIN {X 0,Y 376.048,Z 493.448,A -85,B 0,C 180,E1 -12519.141,E2 -12519.141} C_VEL
LIN {X 0,Y 376.767,Z 487.165,A -85,B 0,C 180,E1 -12520.751,E2 -12520.751} C_VEL
LIN {X 0,Y 377.598,Z 479.3,A -85,B 0,C 180,E1 -12522.36,E2 -12522.36} C_VEL
LIN {X 0,Y 378.622,Z 469.508,A -85,B 0,C 180,E1 -12523.964,E2 -12523.964} C_VEL
LIN {X 0,Y 379.585,Z 460.16,A -85,B 0,C 180,E1 -12525.187,E2 -12525.187} C_VEL
LIN {X 0,Y 380.401,Z 449.033,A -85,B 0,C 180,E1 -12526.365,E2 -12526.365} C_VEL
LIN {X 0,Y 381.335,Z 437.108,A -85,B 0,C 180,E1 -12527.349,E2 -12527.349} C_VEL
LIN {X 0,Y 381.552,Z 430.2,A -85,B 0,C 180,E1 -12527.815,E2 -12527.815} C_VEL
LIN {X 0,Y 378.706,Z 417.903,A -85,B 0,C 180,E1 -12528.636,E2 -12528.636} C_VEL
LIN {X 0,Y 375.065,Z 405.098,A -85,B 0,C 180,E1 -12529.328,E2 -12529.328} C_VEL
LIN {X 0,Y 375.171,Z 401.562,A -85,B 0,C 180,E1 -12532.845,E2 -12532.845} C_VEL
LIN {X 0,Y 374.57,Z 400.786,A -85,B 0,C 180,E1 -12533.734,E2 -12533.734} C_VEL
LIN {X 0,Y 371.751,Z 399.763,A -85,B 0,C 180,E1 -12535.185,E2 -12535.185} C_VEL
LIN {X 0,Y 369.336,Z 398.978,A -85,B 0,C 180,E1 -12536.359,E2 -12536.359} C_VEL
LIN {X 0,Y 368.309,Z 398.283,A -85,B 0,C 180,E1 -12537.265,E2 -12537.265} C_VEL
LIN {X 0,Y 368.233,Z 398.015,A -85,B 0,C 180,E1 -12537.571,E2 -12537.571} C_VEL
LIN {X 0,Y 368.387,Z 394.997,A -85,B 0,C 180,E1 -12541.004,E2 -12541.004} C_VEL
LIN {X 0,Y 368.559,Z 394.578,A -85,B 0,C 180,E1 -12542.962,E2 -12542.962} C_VEL
LIN {X 0,Y 368.857,Z 394.538,A -85,B 0,C 180,E1 -12546.204,E2 -12546.204} C_VEL
LIN {X 0,Y 368.904,Z 394.531,A -85,B 0,C 180,E1 -12548.953,E2 -12548.953} C_VEL
LIN {X 0,Y 368.884,Z 394.534,A -85,B 0,C 180,E1 -12552.01,E2 -12552.01} C_VEL
LIN {X 0,Y 368.883,Z 394.532,A -85,B 0,C 180,E1 -12555.176,E2 -12555.176} C_VEL
LIN {X 0,Y 368.887,Z 394.536,A -85,B 0,C 180,E1 -12558.178,E2 -12558.178} C_VEL
LIN {X 0,Y 368.914,Z 394.528,A -85,B 0,C 180,E1 -12561.359,E2 -12561.359} C_VEL
LIN {X 0,Y 368.941,Z 394.525,A -85,B 0,C 180,E1 -12565.147,E2 -12565.147} C_VEL
LIN {X 0,Y 368.933,Z 394.526,A -85,B 0,C 180,E1 -12569.047,E2 -12569.047} C_VEL
LIN {X 0,Y 368.967,Z 394.522,A -85,B 0,C 180,E1 -12572.797,E2 -12572.797} C_VEL
LIN {X 0,Y 368.938,Z 394.531,A -85,B 0,C 180,E1 -12576.117,E2 -12576.117} C_VEL
LIN {X 0,Y 368.941,Z 394.531,A -85,B 0,C 180,E1 -12579.947,E2 -12579.947} C_VEL
LIN {X 0,Y 368.98,Z 394.521,A -85,B 0,C 180,E1 -12583.399,E2 -12583.399} C_VEL
LIN {X 0,Y 369.062,Z 394.51,A -85,B 0,C 180,E1 -12586.79,E2 -12586.79} C_VEL
LIN {X 0,Y 369.068,Z 394.512,A -85,B 0,C 180,E1 -12590.132,E2 -12590.132} C_VEL
LIN {X 0,Y 369.195,Z 394.496,A -85,B 0,C 180,E1 -12593.442,E2 -12593.442} C_VEL
LIN {X 0,Y 369.321,Z 394.483,A -85,B 0,C 180,E1 -12597.819,E2 -12597.819} C_VEL
LIN {X 0,Y 369.461,Z 394.463,A -85,B 0,C 180,E1 -12600,E2 -12600} C_VEL
LIN {X 0,Y 369.321,Z 394.479,A -85,B 0,C 180,E1 -12602.181,E2 -12602.181} C_VEL
LIN {X 0,Y 369.213,Z 394.491,A -85,B 0,C 180,E1 -12606.558,E2 -12606.558} C_VEL
LIN {X 0,Y 369.144,Z 394.5,A -85,B 0,C 180,E1 -12608.761,E2 -12608.761} C_VEL
LIN {X 0,Y 369.018,Z 394.516,A -85,B 0,C 180,E1 -12612.093,E2 -12612.093} C_VEL
LIN {X 0,Y 369.003,Z 394.523,A -85,B 0,C 180,E1 -12615.465,E2 -12615.465} C_VEL
LIN {X 0,Y 368.962,Z 394.524,A -85,B 0,C 180,E1 -12618.894,E2 -12618.894} C_VEL
LIN {X 0,Y 368.936,Z 394.525,A -85,B 0,C 180,E1 -12622.395,E2 -12622.395} C_VEL
LIN {X 0,Y 369.004,Z 394.517,A -85,B 0,C 180,E1 -12625.98,E2 -12625.98} C_VEL
LIN {X 0,Y 368.918,Z 394.529,A -85,B 0,C 180,E1 -12629.69,E2 -12629.69} C_VEL
LIN {X 0,Y 368.9,Z 394.535,A -85,B 0,C 180,E1 -12633.043,E2 -12633.043} C_VEL
LIN {X 0,Y 368.921,Z 394.527,A -85,B 0,C 180,E1 -12636.197,E2 -12636.197} C_VEL
LIN {X 0,Y 368.907,Z 394.534,A -85,B 0,C 180,E1 -12638.953,E2 -12638.953} C_VEL
LIN {X 0,Y 368.885,Z 394.54,A -85,B 0,C 180,E1 -12642.009,E2 -12642.009} C_VEL
LIN {X 0,Y 368.909,Z 394.566,A -85,B 0,C 180,E1 -12644.33,E2 -12644.33} C_VEL
LIN {X 0,Y 369.97,Z 400.112,A -85,B 0,C 180,E1 -12647.804,E2 -12647.804} C_VEL
LIN {X 0,Y 371.037,Z 406.196,A -85,B 0,C 180,E1 -12651.312,E2 -12651.312} C_VEL
LIN {X 0,Y 371.507,Z 410.1,A -85,B 0,C 180,E1 -12653.423,E2 -12653.423} C_VEL
LIN {X 0,Y 371.003,Z 416.126,A -85,B 0,C 180,E1 -12656.46,E2 -12656.46} C_VEL
LIN {X 0,Y 370.252,Z 423.014,A -85,B 0,C 180,E1 -12659.8,E2 -12659.8} C_VEL
LIN {X 0,Y 369.595,Z 430.524,A -85,B 0,C 180,E1 -12663.345,E2 -12663.345} C_VEL
LIN {X 0,Y 368.926,Z 438.387,A -85,B 0,C 180,E1 -12667.013,E2 -12667.013} C_VEL
LIN {X 0,Y 368.457,Z 445.476,A -85,B 0,C 180,E1 -12670.319,E2 -12670.319} C_VEL
LIN {X 0,Y 370.83,Z 459.245,A -85,B 0,C 180,E1 -12670.914,E2 -12670.914} C_VEL
LIN {X 0,Y 372.469,Z 471.823,A -85,B 0,C 180,E1 -12671.656,E2 -12671.656} C_VEL
LIN {X 0,Y 373.519,Z 481.61,A -85,B 0,C 180,E1 -12672.377,E2 -12672.377} C_VEL
LIN {X 0,Y 372.441,Z 493.938,A -85,B 0,C 180,E1 -12673.416,E2 -12673.416} C_VEL
LIN {X 0,Y 371.303,Z 505.231,A -85,B 0,C 180,E1 -12674.633,E2 -12674.633} C_VEL
LIN {X 0,Y 370.402,Z 515.249,A -85,B 0,C 180,E1 -12676,E2 -12676} C_VEL
LIN {X 0,Y 369.554,Z 523.469,A -85,B 0,C 180,E1 -12677.367,E2 -12677.367} C_VEL
LIN {X 0,Y 368.692,Z 531.538,A -85,B 0,C 180,E1 -12679.011,E2 -12679.011} C_VEL
LIN {X 0,Y 368.166,Z 538.024,A -85,B 0,C 180,E1 -12680.662,E2 -12680.662} C_VEL
LIN {X 0,Y 367.794,Z 543.18,A -85,B 0,C 180,E1 -12682.313,E2 -12682.313} C_VEL
LIN {X 0,Y 367.603,Z 546.852,A -85,B 0,C 180,E1 -12683.807,E2 -12683.807} C_VEL
LIN {X 0,Y 367.519,Z 550.156,A -85,B 0,C 180,E1 -12685.613,E2 -12685.613} C_VEL
LIN {X 0,Y 367.525,Z 552.58,A -85,B 0,C 180,E1 -12687.808,E2 -12687.808} C_VEL
LIN {X 0,Y 367.546,Z 553.197,A -85,B 0,C 180,E1 -12688.904,E2 -12688.904} C_VEL
LIN {X 0,Y 367.538,Z 553.415,A -85,B 0,C 180,E1 -12690,E2 -12690} C_VEL
LIN {X 0,Y 367.546,Z 553.196,A -85,B 0,C 180,E1 -12691.096,E2 -12691.096} C_VEL
LIN {X 0,Y 367.525,Z 552.58,A -85,B 0,C 180,E1 -12692.192,E2 -12692.192} C_VEL
LIN {X 0,Y 367.519,Z 550.155,A -85,B 0,C 180,E1 -12694.387,E2 -12694.387} C_VEL
LIN {X 0,Y 367.598,Z 546.86,A -85,B 0,C 180,E1 -12696.187,E2 -12696.187} C_VEL
LIN {X 0,Y 367.893,Z 541.561,A -85,B 0,C 180,E1 -12698.237,E2 -12698.237} C_VEL
LIN {X 0,Y 368.344,Z 535.987,A -85,B 0,C 180,E1 -12699.888,E2 -12699.888} C_VEL
LIN {X 0,Y 368.935,Z 529.034,A -85,B 0,C 180,E1 -12701.538,E2 -12701.538} C_VEL
LIN {X 0,Y 369.892,Z 520.354,A -85,B 0,C 180,E1 -12703.179,E2 -12703.179} C_VEL
LIN {X 0,Y 370.912,Z 510.093,A -85,B 0,C 180,E1 -12704.735,E2 -12704.735} C_VEL
LIN {X 0,Y 371.757,Z 500.51,A -85,B 0,C 180,E1 -12705.91,E2 -12705.91} C_VEL
LIN {X 0,Y 372.819,Z 489.483,A -85,B 0,C 180,E1 -12706.989,E2 -12706.989} C_VEL
LIN {X 0,Y 373.508,Z 481.555,A -85,B 0,C 180,E1 -12707.623,E2 -12707.623} C_VEL
LIN {X 0,Y 372.275,Z 469.681,A -85,B 0,C 180,E1 -12708.48,E2 -12708.48} C_VEL
LIN {X 0,Y 370.357,Z 456.259,A -85,B 0,C 180,E1 -12709.224,E2 -12709.224} C_VEL
LIN {X 0,Y 368.453,Z 445.402,A -85,B 0,C 180,E1 -12709.681,E2 -12709.681} C_VEL
LIN {X 0,Y 368.937,Z 438.375,A -85,B 0,C 180,E1 -12712.986,E2 -12712.986} C_VEL
LIN {X 0,Y 369.597,Z 430.497,A -85,B 0,C 180,E1 -12716.655,E2 -12716.655} C_VEL
LIN {X 0,Y 370.251,Z 422.965,A -85,B 0,C 180,E1 -12720.2,E2 -12720.2} C_VEL
LIN {X 0,Y 370.994,Z 416.037,A -85,B 0,C 180,E1 -12723.537,E2 -12723.537} C_VEL
LIN {X 0,Y 371.49,Z 411.293,A -85,B 0,C 180,E1 -12725.907,E2 -12725.907} C_VEL
LIN {X 0,Y 371.233,Z 407.425,A -85,B 0,C 180,E1 -12727.971,E2 -12727.971} C_VEL
LIN {X 0,Y 370.145,Z 401.008,A -85,B 0,C 180,E1 -12731.648,E2 -12731.648} C_VEL
LIN {X 0,Y 369.069,Z 395.245,A -85,B 0,C 180,E1 -12735.205,E2 -12735.205} C_VEL
LIN {X 0,Y 368.903,Z 394.544,A -85,B 0,C 180,E1 -12735.831,E2 -12735.831} C_VEL
LIN {X 0,Y 368.914,Z 394.533,A -85,B 0,C 180,E1 -12739.643,E2 -12739.643} C_VEL
LIN {X 0,Y 368.905,Z 394.533,A -85,B 0,C 180,E1 -12743.144,E2 -12743.144} C_VEL
LIN {X 0,Y 368.9,Z 394.532,A -85,B 0,C 180,E1 -12746.462,E2 -12746.462} C_VEL
LIN {X 0,Y 368.931,Z 394.53,A -85,B 0,C 180,E1 -12749.047,E2 -12749.047} C_VEL
LIN {X 0,Y 368.965,Z 394.528,A -85,B 0,C 180,E1 -12752.797,E2 -12752.797} C_VEL
LIN {X 0,Y 368.947,Z 394.525,A -85,B 0,C 180,E1 -12756.113,E2 -12756.113} C_VEL
LIN {X 0,Y 368.939,Z 394.525,A -85,B 0,C 180,E1 -12759.947,E2 -12759.947} C_VEL
LIN {X 0,Y 368.979,Z 394.52,A -85,B 0,C 180,E1 -12763.399,E2 -12763.399} C_VEL
LIN {X 0,Y 369.063,Z 394.513,A -85,B 0,C 180,E1 -12766.79,E2 -12766.79} C_VEL
LIN {X 0,Y 369.075,Z 394.511,A -85,B 0,C 180,E1 -12770.132,E2 -12770.132} C_VEL
LIN {X 0,Y 369.192,Z 394.499,A -85,B 0,C 180,E1 -12772.342,E2 -12772.342} C_VEL
LIN {X 0,Y 369.147,Z 394.504,A -85,B 0,C 180,E1 -12774.538,E2 -12774.538} C_VEL
LIN {X 0,Y 369.32,Z 394.479,A -85,B 0,C 180,E1 -12777.819,E2 -12777.819} C_VEL
LIN {X 0,Y 369.462,Z 394.462,A -85,B 0,C 180,E1 -12780,E2 -12780} C_VEL
LIN {X 0,Y 369.32,Z 394.482,A -85,B 0,C 180,E1 -12782.181,E2 -12782.181} C_VEL
LIN {X 0,Y 369.207,Z 394.494,A -85,B 0,C 180,E1 -12786.625,E2 -12786.625} C_VEL
LIN {X 0,Y 369.14,Z 394.501,A -85,B 0,C 180,E1 -12788.761,E2 -12788.761} C_VEL
LIN {X 0,Y 369.009,Z 394.522,A -85,B 0,C 180,E1 -12792.093,E2 -12792.093} C_VEL
LIN {X 0,Y 369.001,Z 394.518,A -85,B 0,C 180,E1 -12795.465,E2 -12795.465} C_VEL
LIN {X 0,Y 368.969,Z 394.521,A -85,B 0,C 180,E1 -12798.894,E2 -12798.894} C_VEL
LIN {X 0,Y 368.927,Z 394.529,A -85,B 0,C 180,E1 -12802.396,E2 -12802.396} C_VEL
LIN {X 0,Y 369.002,Z 394.523,A -85,B 0,C 180,E1 -12805.98,E2 -12805.98} C_VEL
LIN {X 0,Y 368.917,Z 394.532,A -85,B 0,C 180,E1 -12809.69,E2 -12809.69} C_VEL
LIN {X 0,Y 368.901,Z 394.53,A -85,B 0,C 180,E1 -12813.044,E2 -12813.044} C_VEL
LIN {X 0,Y 368.921,Z 394.53,A -85,B 0,C 180,E1 -12816.197,E2 -12816.197} C_VEL
LIN {X 0,Y 368.907,Z 394.529,A -85,B 0,C 180,E1 -12818.953,E2 -12818.953} C_VEL
LIN {X 0,Y 368.884,Z 394.535,A -85,B 0,C 180,E1 -12822.01,E2 -12822.01} C_VEL
LIN {X 0,Y 368.957,Z 394.524,A -85,B 0,C 180,E1 -12825.187,E2 -12825.187} C_VEL
LIN {X 0,Y 368.947,Z 394.525,A -85,B 0,C 180,E1 -12828.186,E2 -12828.186} C_VEL
LIN {X 0,Y 368.909,Z 394.532,A -85,B 0,C 180,E1 -12831.36,E2 -12831.36} C_VEL
LIN {X 0,Y 368.856,Z 394.539,A -85,B 0,C 180,E1 -12833.796,E2 -12833.796} C_VEL
LIN {X 0,Y 368.539,Z 394.581,A -85,B 0,C 180,E1 -12837.043,E2 -12837.043} C_VEL
LIN {X 0,Y 368.344,Z 395.042,A -85,B 0,C 180,E1 -12839.16,E2 -12839.16} C_VEL
LIN {X 0,Y 368.244,Z 398.18,A -85,B 0,C 180,E1 -12842.739,E2 -12842.739} C_VEL
LIN {X 0,Y 368.157,Z 401.56,A -85,B 0,C 180,E1 -12846.392,E2 -12846.392} C_VEL
LIN {X 0,Y 368.083,Z 405.627,A -85,B 0,C 180,E1 -12850.416,E2 -12850.416} C_VEL
LIN {X 0,Y 371.849,Z 418.988,A -85,B 0,C 180,E1 -12851.14,E2 -12851.14} C_VEL
LIN {X 0,Y 374.565,Z 430.389,A -85,B 0,C 180,E1 -12851.927,E2 -12851.927} C_VEL
LIN {X 0,Y 374.767,Z 434.177,A -85,B 0,C 180,E1 -12852.195,E2 -12852.195} C_VEL
LIN {X 0,Y 373.952,Z 445.449,A -85,B 0,C 180,E1 -12853.064,E2 -12853.064} C_VEL
LIN {X 0,Y 373.157,Z 455.654,A -85,B 0,C 180,E1 -12854.062,E2 -12854.062} C_VEL
LIN {X 0,Y 372.206,Z 465.384,A -85,B 0,C 180,E1 -12855.232,E2 -12855.232} C_VEL
LIN {X 0,Y 371.253,Z 474.524,A -85,B 0,C 180,E1 -12856.591,E2 -12856.591} C_VEL
LIN {X 0,Y 370.255,Z 483.395,A -85,B 0,C 180,E1 -12858.226,E2 -12858.226} C_VEL
LIN {X 0,Y 369.446,Z 490.531,A -85,B 0,C 180,E1 -12859.865,E2 -12859.865} C_VEL
LIN {X 0,Y 368.902,Z 495.341,A -85,B 0,C 180,E1 -12861.234,E2 -12861.234} C_VEL
LIN {X 0,Y 368.488,Z 499.42,A -85,B 0,C 180,E1 -12862.648,E2 -12862.648} C_VEL
LIN {X 0,Y 367.997,Z 503.587,A -85,B 0,C 180,E1 -12864.521,E2 -12864.521} C_VEL
LIN {X 0,Y 367.932,Z 505.425,A -85,B 0,C 180,E1 -12865.618,E2 -12865.618} C_VEL
LIN {X 0,Y 367.913,Z 506.807,A -85,B 0,C 180,E1 -12866.715,E2 -12866.715} C_VEL
LIN {X 0,Y 367.636,Z 508.411,A -85,B 0,C 180,E1 -12868.905,E2 -12868.905} C_VEL
LIN {X 0,Y 367.61,Z 508.642,A -85,B 0,C 180,E1 -12870,E2 -12870} C_VEL
LIN {X 0,Y 367.751,Z 507.868,A -85,B 0,C 180,E1 -12872.191,E2 -12872.191} C_VEL
LIN {X 0,Y 367.909,Z 506.904,A -85,B 0,C 180,E1 -12873.285,E2 -12873.285} C_VEL
LIN {X 0,Y 367.93,Z 505.565,A -85,B 0,C 180,E1 -12874.382,E2 -12874.382} C_VEL
LIN {X 0,Y 368.136,Z 502.723,A -85,B 0,C 180,E1 -12876.027,E2 -12876.027} C_VEL
LIN {X 0,Y 368.532,Z 498.861,A -85,B 0,C 180,E1 -12877.672,E2 -12877.672} C_VEL
LIN {X 0,Y 369.067,Z 493.877,A -85,B 0,C 180,E1 -12879.315,E2 -12879.315} C_VEL
LIN {X 0,Y 369.811,Z 487.594,A -85,B 0,C 180,E1 -12880.955,E2 -12880.955} C_VEL
LIN {X 0,Y 370.691,Z 479.728,A -85,B 0,C 180,E1 -12882.594,E2 -12882.594} C_VEL
LIN {X 0,Y 371.759,Z 469.936,A -85,B 0,C 180,E1 -12884.227,E2 -12884.227} C_VEL
LIN {X 0,Y 372.744,Z 460.69,A -85,B 0,C 180,E1 -12885.46,E2 -12885.46} C_VEL
LIN {X 0,Y 373.613,Z 449.459,A -85,B 0,C 180,E1 -12886.671,E2 -12886.671} C_VEL
LIN {X 0,Y 374.572,Z 437.653,A -85,B 0,C 180,E1 -12887.662,E2 -12887.662} C_VEL
LIN {X 0,Y 374.712,Z 431.117,A -85,B 0,C 180,E1 -12888.121,E2 -12888.121} C_VEL
LIN {X 0,Y 371.669,Z 418.208,A -85,B 0,C 180,E1 -12889.009,E2 -12889.009} C_VEL
LIN {X 0,Y 368.048,Z 405.527,A -85,B 0,C 180,E1 -12889.707,E2 -12889.707} C_VEL
LIN {X 0,Y 368.17,Z 401.651,A -85,B 0,C 180,E1 -12893.633,E2 -12893.633} C_VEL
LIN {X 0,Y 368.232,Z 398.295,A -85,B 0,C 180,E1 -12897.262,E2 -12897.262} C_VEL
LIN {X 0,Y 368.233,Z 398.015,A -85,B 0,C 180,E1 -12897.571,E2 -12897.571} C_VEL
LIN {X 0,Y 367.585,Z 397.287,A -85,B 0,C 180,E1 -12898.477,E2 -12898.477} C_VEL
LIN {X 0,Y 364.762,Z 396.35,A -85,B 0,C 180,E1 -12899.958,E2 -12899.958} C_VEL
LIN {X 0,Y 362.411,Z 395.746,A -85,B 0,C 180,E1 -12901.159,E2 -12901.159} C_VEL
LIN {X 0,Y 361.471,Z 395.488,A -85,B 0,C 180,E1 -12902.089,E2 -12902.089} C_VEL
LIN {X 0,Y 361.432,Z 395.463,A -85,B 0,C 180,E1 -12902.403,E2 -12902.403} C_VEL
LIN {X 0,Y 361.749,Z 395.421,A -85,B 0,C 180,E1 -12905.651,E2 -12905.651} C_VEL
LIN {X 0,Y 361.871,Z 395.407,A -85,B 0,C 180,E1 -12909.026,E2 -12909.026} C_VEL
LIN {X 0,Y 361.839,Z 395.412,A -85,B 0,C 180,E1 -12912.829,E2 -12912.829} C_VEL
LIN {X 0,Y 361.821,Z 395.414,A -85,B 0,C 180,E1 -12915.947,E2 -12915.947} C_VEL
LIN {X 0,Y 361.84,Z 395.409,A -85,B 0,C 180,E1 -12919.245,E2 -12919.245} C_VEL
LIN {X 0,Y 361.875,Z 395.406,A -85,B 0,C 180,E1 -12922.775,E2 -12922.775} C_VEL
LIN {X 0,Y 361.859,Z 395.408,A -85,B 0,C 180,E1 -12925.72,E2 -12925.72} C_VEL
LIN {X 0,Y 361.877,Z 395.406,A -85,B 0,C 180,E1 -12929.672,E2 -12929.672} C_VEL
LIN {X 0,Y 361.958,Z 395.395,A -85,B 0,C 180,E1 -12933.475,E2 -12933.475} C_VEL
LIN {X 0,Y 361.883,Z 395.404,A -85,B 0,C 180,E1 -12937.144,E2 -12937.144} C_VEL
LIN {X 0,Y 361.916,Z 395.4,A -85,B 0,C 180,E1 -12940.724,E2 -12940.724} C_VEL
LIN {X 0,Y 361.937,Z 395.397,A -85,B 0,C 180,E1 -12943.066,E2 -12943.066} C_VEL
LIN {X 0,Y 362.003,Z 395.39,A -85,B 0,C 180,E1 -12946.528,E2 -12946.528} C_VEL
LIN {X 0,Y 362.033,Z 395.391,A -85,B 0,C 180,E1 -12949.938,E2 -12949.938} C_VEL
LIN {X 0,Y 362.156,Z 395.371,A -85,B 0,C 180,E1 -12953.313,E2 -12953.313} C_VEL
LIN {X 0,Y 362.285,Z 395.36,A -85,B 0,C 180,E1 -12957.776,E2 -12957.776} C_VEL
LIN {X 0,Y 362.431,Z 395.339,A -85,B 0,C 180,E1 -12960,E2 -12960} C_VEL
LIN {X 0,Y 362.285,Z 395.355,A -85,B 0,C 180,E1 -12962.223,E2 -12962.223} C_VEL
LIN {X 0,Y 362.177,Z 395.367,A -85,B 0,C 180,E1 -12966.686,E2 -12966.686} C_VEL
LIN {X 0,Y 362.08,Z 395.38,A -85,B 0,C 180,E1 -12968.933,E2 -12968.933} C_VEL
LIN {X 0,Y 361.971,Z 395.393,A -85,B 0,C 180,E1 -12972.332,E2 -12972.332} C_VEL
LIN {X 0,Y 361.967,Z 395.393,A -85,B 0,C 180,E1 -12974.62,E2 -12974.62} C_VEL
LIN {X 0,Y 361.96,Z 395.395,A -85,B 0,C 180,E1 -12978.099,E2 -12978.099} C_VEL
LIN {X 0,Y 361.896,Z 395.405,A -85,B 0,C 180,E1 -12981.653,E2 -12981.653} C_VEL
LIN {X 0,Y 361.932,Z 395.404,A -85,B 0,C 180,E1 -12985.29,E2 -12985.29} C_VEL
LIN {X 0,Y 361.912,Z 395.402,A -85,B 0,C 180,E1 -12987.779,E2 -12987.779} C_VEL
LIN {X 0,Y 361.841,Z 395.411,A -85,B 0,C 180,E1 -12991.629,E2 -12991.629} C_VEL
LIN {X 0,Y 361.878,Z 395.409,A -85,B 0,C 180,E1 -12995.345,E2 -12995.345} C_VEL
LIN {X 0,Y 361.874,Z 395.411,A -85,B 0,C 180,E1 -12999.027,E2 -12999.027} C_VEL
LIN {X 0,Y 361.839,Z 395.415,A -85,B 0,C 180,E1 -13002.829,E2 -13002.829} C_VEL
LIN {X 0,Y 361.884,Z 395.553,A -85,B 0,C 180,E1 -13003.964,E2 -13003.964} C_VEL
LIN {X 0,Y 362.877,Z 400.883,A -85,B 0,C 180,E1 -13007.389,E2 -13007.389} C_VEL
LIN {X 0,Y 363.842,Z 406.267,A -85,B 0,C 180,E1 -13010.592,E2 -13010.592} C_VEL
LIN {X 0,Y 364.497,Z 411.096,A -85,B 0,C 180,E1 -13013.293,E2 -13013.293} C_VEL
LIN {X 0,Y 364.05,Z 416.552,A -85,B 0,C 180,E1 -13016.111,E2 -13016.111} C_VEL
LIN {X 0,Y 363.328,Z 422.682,A -85,B 0,C 180,E1 -13019.162,E2 -13019.162} C_VEL
LIN {X 0,Y 362.742,Z 429.119,A -85,B 0,C 180,E1 -13022.29,E2 -13022.29} C_VEL
LIN {X 0,Y 362.024,Z 436.731,A -85,B 0,C 180,E1 -13025.941,E2 -13025.941} C_VEL
LIN {X 0,Y 361.45,Z 444.824,A -85,B 0,C 180,E1 -13029.81,E2 -13029.81} C_VEL
LIN {X 0,Y 361.427,Z 445.052,A -85,B 0,C 180,E1 -13029.92,E2 -13029.92} C_VEL
LIN {X 0,Y 363.838,Z 458.941,A -85,B 0,C 180,E1 -13030.539,E2 -13030.539} C_VEL
LIN {X 0,Y 365.564,Z 472.192,A -85,B 0,C 180,E1 -13031.348,E2 -13031.348} C_VEL
LIN {X 0,Y 366.649,Z 482.46,A -85,B 0,C 180,E1 -13032.14,E2 -13032.14} C_VEL
LIN {X 0,Y 365.475,Z 494.935,A -85,B 0,C 180,E1 -13033.235,E2 -13033.235} C_VEL
LIN {X 0,Y 364.418,Z 504.798,A -85,B 0,C 180,E1 -13034.336,E2 -13034.336} C_VEL
LIN {X 0,Y 363.494,Z 514.818,A -85,B 0,C 180,E1 -13035.728,E2 -13035.728} C_VEL
LIN {X 0,Y 362.409,Z 524.532,A -85,B 0,C 180,E1 -13037.399,E2 -13037.399} C_VEL
LIN {X 0,Y 361.589,Z 532.276,A -85,B 0,C 180,E1 -13039.076,E2 -13039.076} C_VEL
LIN {X 0,Y 360.971,Z 539.427,A -85,B 0,C 180,E1 -13041.039,E2 -13041.039} C_VEL
LIN {X 0,Y 360.679,Z 544.195,A -85,B 0,C 180,E1 -13042.723,E2 -13042.723} C_VEL
LIN {X 0,Y 360.478,Z 547.84,A -85,B 0,C 180,E1 -13044.406,E2 -13044.406} C_VEL
LIN {X 0,Y 360.451,Z 549.725,A -85,B 0,C 180,E1 -13045.527,E2 -13045.527} C_VEL
LIN {X 0,Y 360.428,Z 552.148,A -85,B 0,C 180,E1 -13047.765,E2 -13047.765} C_VEL
LIN {X 0,Y 360.483,Z 552.767,A -85,B 0,C 180,E1 -13048.883,E2 -13048.883} C_VEL
LIN {X 0,Y 360.473,Z 552.985,A -85,B 0,C 180,E1 -13050,E2 -13050} C_VEL
LIN {X 0,Y 360.483,Z 552.766,A -85,B 0,C 180,E1 -13051.117,E2 -13051.117} C_VEL
LIN {X 0,Y 360.428,Z 552.147,A -85,B 0,C 180,E1 -13052.235,E2 -13052.235} C_VEL
LIN {X 0,Y 360.45,Z 549.723,A -85,B 0,C 180,E1 -13054.473,E2 -13054.473} C_VEL
LIN {X 0,Y 360.527,Z 546.693,A -85,B 0,C 180,E1 -13056.184,E2 -13056.184} C_VEL
LIN {X 0,Y 360.719,Z 542.734,A -85,B 0,C 180,E1 -13057.839,E2 -13057.839} C_VEL
LIN {X 0,Y 361.225,Z 536.571,A -85,B 0,C 180,E1 -13059.802,E2 -13059.802} C_VEL
LIN {X 0,Y 361.828,Z 529.843,A -85,B 0,C 180,E1 -13061.484,E2 -13061.484} C_VEL
LIN {X 0,Y 362.787,Z 521.515,A -85,B 0,C 180,E1 -13063.157,E2 -13063.157} C_VEL
LIN {X 0,Y 363.71,Z 512.981,A -85,B 0,C 180,E1 -13064.549,E2 -13064.549} C_VEL
LIN {X 0,Y 364.528,Z 503.617,A -85,B 0,C 180,E1 -13065.803,E2 -13065.803} C_VEL
LIN {X 0,Y 365.732,Z 492.026,A -85,B 0,C 180,E1 -13067.041,E2 -13067.041} C_VEL
LIN {X 0,Y 366.629,Z 482.395,A -85,B 0,C 180,E1 -13067.861,E2 -13067.861} C_VEL
LIN {X 0,Y 365.369,Z 470.038,A -85,B 0,C 180,E1 -13068.793,E2 -13068.793} C_VEL
LIN {X 0,Y 363.559,Z 456.896,A -85,B 0,C 180,E1 -13069.555,E2 -13069.555} C_VEL
LIN {X 0,Y 361.424,Z 444.986,A -85,B 0,C 180,E1 -13070.079,E2 -13070.079} C_VEL
LIN {X 0,Y 361.919,Z 437.977,A -85,B 0,C 180,E1 -13073.458,E2 -13073.458} C_VEL
LIN {X 0,Y 362.571,Z 430.742,A -85,B 0,C 180,E1 -13076.918,E2 -13076.918} C_VEL
LIN {X 0,Y 363.218,Z 423.939,A -85,B 0,C 180,E1 -13080.204,E2 -13080.204} C_VEL
LIN {X 0,Y 363.912,Z 417.577,A -85,B 0,C 180,E1 -13083.321,E2 -13083.321} C_VEL
LIN {X 0,Y 364.472,Z 412.488,A -85,B 0,C 180,E1 -13085.916,E2 -13085.916} C_VEL
LIN {X 0,Y 364.201,Z 408.418,A -85,B 0,C 180,E1 -13088.134,E2 -13088.134} C_VEL
LIN {X 0,Y 363.34,Z 403.295,A -85,B 0,C 180,E1 -13091.121,E2 -13091.121} C_VEL
LIN {X 0,Y 362.229,Z 397.123,A -85,B 0,C 180,E1 -13094.978,E2 -13094.978} C_VEL
LIN {X 0,Y 361.866,Z 395.416,A -85,B 0,C 180,E1 -13096.24,E2 -13096.24} C_VEL
LIN {X 0,Y 361.858,Z 395.415,A -85,B 0,C 180,E1 -13100.139,E2 -13100.139} C_VEL
LIN {X 0,Y 361.871,Z 395.411,A -85,B 0,C 180,E1 -13102.982,E2 -13102.982} C_VEL
LIN {X 0,Y 361.862,Z 395.411,A -85,B 0,C 180,E1 -13106.63,E2 -13106.63} C_VEL
LIN {X 0,Y 361.875,Z 395.405,A -85,B 0,C 180,E1 -13109.672,E2 -13109.672} C_VEL
LIN {X 0,Y 361.956,Z 395.395,A -85,B 0,C 180,E1 -13113.475,E2 -13113.475} C_VEL
LIN {X 0,Y 361.893,Z 395.405,A -85,B 0,C 180,E1 -13117.145,E2 -13117.145} C_VEL
LIN {X 0,Y 361.909,Z 395.406,A -85,B 0,C 180,E1 -13120.724,E2 -13120.724} C_VEL
LIN {X 0,Y 361.936,Z 395.399,A -85,B 0,C 180,E1 -13123.066,E2 -13123.066} C_VEL
LIN {X 0,Y 362.004,Z 395.395,A -85,B 0,C 180,E1 -13126.528,E2 -13126.528} C_VEL
LIN {X 0,Y 362.039,Z 395.386,A -85,B 0,C 180,E1 -13129.938,E2 -13129.938} C_VEL
LIN {X 0,Y 362.155,Z 395.373,A -85,B 0,C 180,E1 -13132.193,E2 -13132.193} C_VEL
LIN {X 0,Y 362.121,Z 395.381,A -85,B 0,C 180,E1 -13134.431,E2 -13134.431} C_VEL
LIN {X 0,Y 362.284,Z 395.355,A -85,B 0,C 180,E1 -13137.777,E2 -13137.777} C_VEL
LIN {X 0,Y 362.431,Z 395.338,A -85,B 0,C 180,E1 -13140,E2 -13140} C_VEL
LIN {X 0,Y 362.283,Z 395.359,A -85,B 0,C 180,E1 -13142.224,E2 -13142.224} C_VEL
LIN {X 0,Y 362.176,Z 395.369,A -85,B 0,C 180,E1 -13146.686,E2 -13146.686} C_VEL
LIN {X 0,Y 362.077,Z 395.38,A -85,B 0,C 180,E1 -13148.933,E2 -13148.933} C_VEL
LIN {X 0,Y 361.963,Z 395.398,A -85,B 0,C 180,E1 -13152.332,E2 -13152.332} C_VEL
LIN {X 0,Y 361.965,Z 395.395,A -85,B 0,C 180,E1 -13154.62,E2 -13154.62} C_VEL
LIN {X 0,Y 361.96,Z 395.401,A -85,B 0,C 180,E1 -13158.099,E2 -13158.099} C_VEL
LIN {X 0,Y 361.883,Z 395.406,A -85,B 0,C 180,E1 -13161.654,E2 -13161.654} C_VEL
LIN {X 0,Y 361.93,Z 395.399,A -85,B 0,C 180,E1 -13165.29,E2 -13165.29} C_VEL
LIN {X 0,Y 361.911,Z 395.405,A -85,B 0,C 180,E1 -13167.779,E2 -13167.779} C_VEL
LIN {X 0,Y 361.84,Z 395.413,A -85,B 0,C 180,E1 -13171.629,E2 -13171.629} C_VEL
LIN {X 0,Y 361.877,Z 395.406,A -85,B 0,C 180,E1 -13175.345,E2 -13175.345} C_VEL
LIN {X 0,Y 361.873,Z 395.405,A -85,B 0,C 180,E1 -13179.027,E2 -13179.027} C_VEL
LIN {X 0,Y 361.841,Z 395.409,A -85,B 0,C 180,E1 -13182.828,E2 -13182.828} C_VEL
LIN {X 0,Y 361.914,Z 395.404,A -85,B 0,C 180,E1 -13185.931,E2 -13185.931} C_VEL
LIN {X 0,Y 361.908,Z 395.403,A -85,B 0,C 180,E1 -13189.232,E2 -13189.232} C_VEL
LIN {X 0,Y 361.839,Z 395.41,A -85,B 0,C 180,E1 -13192.978,E2 -13192.978} C_VEL
LIN {X 0,Y 361.632,Z 395.441,A -85,B 0,C 180,E1 -13195.695,E2 -13195.695} C_VEL
LIN {X 0,Y 361.31,Z 395.706,A -85,B 0,C 180,E1 -13198.856,E2 -13198.856} C_VEL
LIN {X 0,Y 361.232,Z 398.559,A -85,B 0,C 180,E1 -13202.164,E2 -13202.164} C_VEL
LIN {X 0,Y 361.121,Z 401.94,A -85,B 0,C 180,E1 -13205.877,E2 -13205.877} C_VEL
LIN {X 0,Y 361.032,Z 406.026,A -85,B 0,C 180,E1 -13210.008,E2 -13210.008} C_VEL
LIN {X 0,Y 365.065,Z 420.189,A -85,B 0,C 180,E1 -13210.812,E2 -13210.812} C_VEL
LIN {X 0,Y 367.958,Z 432.569,A -85,B 0,C 180,E1 -13211.705,E2 -13211.705} C_VEL
LIN {X 0,Y 367.789,Z 438.218,A -85,B 0,C 180,E1 -13212.114,E2 -13212.114} C_VEL
LIN {X 0,Y 366.837,Z 450.302,A -85,B 0,C 180,E1 -13213.156,E2 -13213.156} C_VEL
LIN {X 0,Y 365.875,Z 461.567,A -85,B 0,C 180,E1 -13214.4,E2 -13214.4} C_VEL
LIN {X 0,Y 364.759,Z 471.505,A -85,B 0,C 180,E1 -13215.779,E2 -13215.779} C_VEL
LIN {X 0,Y 363.831,Z 479.634,A -85,B 0,C 180,E1 -13217.165,E2 -13217.165} C_VEL
LIN {X 0,Y 362.931,Z 487.589,A -85,B 0,C 180,E1 -13218.834,E2 -13218.834} C_VEL
LIN {X 0,Y 362.092,Z 493.978,A -85,B 0,C 180,E1 -13220.504,E2 -13220.504} C_VEL
LIN {X 0,Y 361.456,Z 500.045,A -85,B 0,C 180,E1 -13222.581,E2 -13222.581} C_VEL
LIN {X 0,Y 360.956,Z 504.018,A -85,B 0,C 180,E1 -13224.413,E2 -13224.413} C_VEL
LIN {X 0,Y 360.855,Z 505.858,A -85,B 0,C 180,E1 -13225.532,E2 -13225.532} C_VEL
LIN {X 0,Y 360.858,Z 507.238,A -85,B 0,C 180,E1 -13226.651,E2 -13226.651} C_VEL
LIN {X 0,Y 360.571,Z 508.841,A -85,B 0,C 180,E1 -13228.883,E2 -13228.883} C_VEL
LIN {X 0,Y 360.543,Z 509.073,A -85,B 0,C 180,E1 -13230,E2 -13230} C_VEL
LIN {X 0,Y 360.693,Z 508.298,A -85,B 0,C 180,E1 -13232.233,E2 -13232.233} C_VEL
LIN {X 0,Y 360.835,Z 507.335,A -85,B 0,C 180,E1 -13233.35,E2 -13233.35} C_VEL
LIN {X 0,Y 360.853,Z 505.996,A -85,B 0,C 180,E1 -13234.468,E2 -13234.468} C_VEL
LIN {X 0,Y 361.108,Z 503.152,A -85,B 0,C 180,E1 -13236.145,E2 -13236.145} C_VEL
LIN {X 0,Y 361.513,Z 499.291,A -85,B 0,C 180,E1 -13237.821,E2 -13237.821} C_VEL
LIN {X 0,Y 362.076,Z 494.307,A -85,B 0,C 180,E1 -13239.497,E2 -13239.497} C_VEL
LIN {X 0,Y 362.863,Z 488.023,A -85,B 0,C 180,E1 -13241.168,E2 -13241.168} C_VEL
LIN {X 0,Y 363.788,Z 480.156,A -85,B 0,C 180,E1 -13242.837,E2 -13242.837} C_VEL
LIN {X 0,Y 364.897,Z 470.364,A -85,B 0,C 180,E1 -13244.5,E2 -13244.5} C_VEL
LIN {X 0,Y 365.987,Z 460.222,A -85,B 0,C 180,E1 -13245.863,E2 -13245.863} C_VEL
LIN {X 0,Y 366.837,Z 449.885,A -85,B 0,C 180,E1 -13246.988,E2 -13246.988} C_VEL
LIN {X 0,Y 367.829,Z 438.179,A -85,B 0,C 180,E1 -13247.989,E2 -13247.989} C_VEL
LIN {X 0,Y 368.061,Z 433.097,A -85,B 0,C 180,E1 -13248.353,E2 -13248.353} C_VEL
LIN {X 0,Y 365.272,Z 420.848,A -85,B 0,C 180,E1 -13249.247,E2 -13249.247} C_VEL
LIN {X 0,Y 361.443,Z 407.813,A -85,B 0,C 180,E1 -13250.005,E2 -13250.005} C_VEL
LIN {X 0,Y 360.994,Z 405.96,A -85,B 0,C 180,E1 -13250.104,E2 -13250.104} C_VEL
LIN {X 0,Y 361.122,Z 402.05,A -85,B 0,C 180,E1 -13254.123,E2 -13254.123} C_VEL
LIN {X 0,Y 361.22,Z 398.666,A -85,B 0,C 180,E1 -13257.837,E2 -13257.837} C_VEL
LIN {X 0,Y 361.345,Z 395.789,A -85,B 0,C 180,E1 -13261.154,E2 -13261.154} C_VEL
LIN {X 0,Y 361.432,Z 395.463,A -85,B 0,C 180,E1 -13262.403,E2 -13262.403} C_VEL
LIN {X 0,Y 360.882,Z 395.535,A -85,B 0,C 180,E1 -13263.335,E2 -13263.335} C_VEL
LIN {X 0,Y 358.145,Z 395.873,A -85,B 0,C 180,E1 -13264.855,E2 -13264.855} C_VEL
LIN {X 0,Y 355.797,Z 396.164,A -85,B 0,C 180,E1 -13266.084,E2 -13266.084} C_VEL
LIN {X 0,Y 354.826,Z 396.285,A -85,B 0,C 180,E1 -13267.033,E2 -13267.033} C_VEL
LIN {X 0,Y 354.769,Z 396.29,A -85,B 0,C 180,E1 -13267.355,E2 -13267.355} C_VEL
LIN {X 0,Y 354.827,Z 396.283,A -85,B 0,C 180,E1 -13269.424,E2 -13269.424} C_VEL
LIN {X 0,Y 354.791,Z 396.289,A -85,B 0,C 180,E1 -13272.867,E2 -13272.867} C_VEL
LIN {X 0,Y 354.77,Z 396.293,A -85,B 0,C 180,E1 -13276.104,E2 -13276.104} C_VEL
LIN {X 0,Y 354.792,Z 396.287,A -85,B 0,C 180,E1 -13279.179,E2 -13279.179} C_VEL
LIN {X 0,Y 354.816,Z 396.289,A -85,B 0,C 180,E1 -13282.401,E2 -13282.401} C_VEL
LIN {X 0,Y 354.816,Z 396.284,A -85,B 0,C 180,E1 -13284.941,E2 -13284.941} C_VEL
LIN {X 0,Y 354.797,Z 396.29,A -85,B 0,C 180,E1 -13288.405,E2 -13288.405} C_VEL
LIN {X 0,Y 354.85,Z 396.281,A -85,B 0,C 180,E1 -13291.619,E2 -13291.619} C_VEL
LIN {X 0,Y 354.902,Z 396.279,A -85,B 0,C 180,E1 -13294.173,E2 -13294.173} C_VEL
LIN {X 0,Y 354.819,Z 396.288,A -85,B 0,C 180,E1 -13297.893,E2 -13297.893} C_VEL
LIN {X 0,Y 354.927,Z 396.276,A -85,B 0,C 180,E1 -13301.892,E2 -13301.892} C_VEL
LIN {X 0,Y 354.947,Z 396.273,A -85,B 0,C 180,E1 -13305.981,E2 -13305.981} C_VEL
LIN {X 0,Y 354.98,Z 396.269,A -85,B 0,C 180,E1 -13309.736,E2 -13309.736} C_VEL
LIN {X 0,Y 355.119,Z 396.247,A -85,B 0,C 180,E1 -13313.18,E2 -13313.18} C_VEL
LIN {X 0,Y 355.248,Z 396.237,A -85,B 0,C 180,E1 -13317.732,E2 -13317.732} C_VEL
LIN {X 0,Y 355.401,Z 396.215,A -85,B 0,C 180,E1 -13320,E2 -13320} C_VEL
LIN {X 0,Y 355.248,Z 396.232,A -85,B 0,C 180,E1 -13322.268,E2 -13322.268} C_VEL
LIN {X 0,Y 355.143,Z 396.244,A -85,B 0,C 180,E1 -13326.819,E2 -13326.819} C_VEL
LIN {X 0,Y 355.021,Z 396.261,A -85,B 0,C 180,E1 -13329.112,E2 -13329.112} C_VEL
LIN {X 0,Y 354.931,Z 396.27,A -85,B 0,C 180,E1 -13332.581,E2 -13332.581} C_VEL
LIN {X 0,Y 354.894,Z 396.275,A -85,B 0,C 180,E1 -13336.096,E2 -13336.096} C_VEL
LIN {X 0,Y 354.905,Z 396.273,A -85,B 0,C 180,E1 -13338.472,E2 -13338.472} C_VEL
LIN {X 0,Y 354.838,Z 396.282,A -85,B 0,C 180,E1 -13342.106,E2 -13342.106} C_VEL
LIN {X 0,Y 354.903,Z 396.275,A -85,B 0,C 180,E1 -13345.827,E2 -13345.827} C_VEL
LIN {X 0,Y 354.821,Z 396.286,A -85,B 0,C 180,E1 -13349.682,E2 -13349.682} C_VEL
LIN {X 0,Y 354.809,Z 396.287,A -85,B 0,C 180,E1 -13353.702,E2 -13353.702} C_VEL
LIN {X 0,Y 354.801,Z 396.287,A -85,B 0,C 180,E1 -13356.459,E2 -13356.459} C_VEL
LIN {X 0,Y 354.827,Z 396.287,A -85,B 0,C 180,E1 -13359.423,E2 -13359.423} C_VEL
LIN {X 0,Y 354.815,Z 396.387,A -85,B 0,C 180,E1 -13363.468,E2 -13363.468} C_VEL
LIN {X 0,Y 355.819,Z 401.655,A -85,B 0,C 180,E1 -13366.954,E2 -13366.954} C_VEL
LIN {X 0,Y 356.771,Z 406.931,A -85,B 0,C 180,E1 -13370.198,E2 -13370.198} C_VEL
LIN {X 0,Y 357.481,Z 412.06,A -85,B 0,C 180,E1 -13373.14,E2 -13373.14} C_VEL
LIN {X 0,Y 357.101,Z 416.985,A -85,B 0,C 180,E1 -13375.75,E2 -13375.75} C_VEL
LIN {X 0,Y 356.466,Z 422.423,A -85,B 0,C 180,E1 -13378.538,E2 -13378.538} C_VEL
LIN {X 0,Y 355.678,Z 429.994,A -85,B 0,C 180,E1 -13382.313,E2 -13382.313} C_VEL
LIN {X 0,Y 354.928,Z 437.752,A -85,B 0,C 180,E1 -13386.129,E2 -13386.129} C_VEL
LIN {X 0,Y 354.402,Z 444.625,A -85,B 0,C 180,E1 -13389.504,E2 -13389.504} C_VEL
LIN {X 0,Y 356.866,Z 458.444,A -85,B 0,C 180,E1 -13390.141,E2 -13390.141} C_VEL
LIN {X 0,Y 358.615,Z 471.752,A -85,B 0,C 180,E1 -13390.973,E2 -13390.973} C_VEL
LIN {X 0,Y 359.725,Z 483.804,A -85,B 0,C 180,E1 -13391.931,E2 -13391.931} C_VEL
LIN {X 0,Y 358.67,Z 494.506,A -85,B 0,C 180,E1 -13392.907,E2 -13392.907} C_VEL
LIN {X 0,Y 357.558,Z 504.367,A -85,B 0,C 180,E1 -13394.027,E2 -13394.027} C_VEL
LIN {X 0,Y 356.589,Z 514.386,A -85,B 0,C 180,E1 -13395.446,E2 -13395.446} C_VEL
LIN {X 0,Y 355.461,Z 524.1,A -85,B 0,C 180,E1 -13397.148,E2 -13397.148} C_VEL
LIN {X 0,Y 354.556,Z 531.841,A -85,B 0,C 180,E1 -13398.856,E2 -13398.856} C_VEL
LIN {X 0,Y 354.087,Z 537.157,A -85,B 0,C 180,E1 -13400.287,E2 -13400.287} C_VEL
